// TwinCAT 3 PLC project RoboTelRuntime
// Company: Leibniz-Institut fuer Astrophysik Potsdam
// Author: Joerg Weingrill
// ProgramVersion: 3.1.4023.0
// libraries:
//   Tc2_Math, * (Beckhoff Automation GmbH)
//   Tc2_MC2, * (Beckhoff Automation GmbH)
//   Tc2_MC2_Drive, * (Beckhoff Automation GmbH)
//   Tc2_ModbusRTU, * (Beckhoff Automation GmbH)
//   Tc2_NC, * (Beckhoff Automation GmbH)
//   Tc2_Standard, * (Beckhoff Automation GmbH)
//   Tc2_System, * (Beckhoff Automation GmbH)
//   Tc2_Utilities, * (Beckhoff Automation GmbH)
//   Tc3_IotBase, * (Beckhoff Automation GmbH)
//   Tc3_Module, * (Beckhoff Automation GmbH)
//   PS_DcUpsEC,2.0,Phoenix Contact GmbH & Co.KG
// project tree:
//   DUTs/ E_TCSCommand.TcDUT, E_TCSErrors.TcDUT, E_TelescopeMode.TcDUT, ST_DomeStruct.TcDUT
//   / GlobalTextList.TcGTLO, PlcTask.TcTTO, Visualisierungsmanager.TcVMO (not stored)
//   GVLs/ GVL_Auxiliary.TcGVL, GVL_Dome.TcGVL, GVL_Environment.TcGVL, GVL_FilterWheel.TcGVL, GVL_pendant_control.TcGVL, GVL_Hydraulics.TcGVL, GVL_Safety.TcGVL, GVL_Telescope.TcGVL, GVL_Main.TcGVL
//   POUs/ AuxiliaryControl.TcPOU, CoverControl.TcPOU, DerotatorControl.TcPOU, DomeControl.TcPOU, DomeLowLevelControl.TcPOU, ElevationControl.TcPOU, AzimuthElevationControl.TcPOU, Environment.TcPOU, FanControl.TcPOU, FilterWheelControl.TcPOU, FocusControl.TcPOU, HydraulicsControl.TcPOU, MAIN.TcPOU, NasmythControl.TcPOU, PendantControl.TcPOU, SafetyHandling.TcPOU, TelescopeAuxiliary.TcPOU, TelescopeControl.TcPOU, Transformer.TcPOU
//   POUs/FunctionBlocks/ CO_ABERRATION.TcPOU, CO_REFRACT.TcPOU, FB_ALTAZ2HADEC.TcPOU, FB_AstroClock.TcPOU, FB_Axis2.TcPOU, FB_BLINK.TcPOU, FB_ButtonEnable.TcPOU, FB_CO_NUTATE.TcPOU, FB_EQ2HOR2.TcPOU, FB_EventLog.TcPOU, FB_HOR2EQ.TcPOU, FB_LightTimer.TcPOU, FB_MOONPOS.TcPOU, FB_MQTTCommunication.TcPOU, FB_NUTATE.TcPOU, FB_PRECESS.TcPOU, FB_SUNPOS.TcPOU, FB_TimeAverage.TcPOU, FB_Timer.TcPOU, FB_TONTP.TcPOU, FB_InfluxMessage.TcPOU, TIMER.TcPOU
//   POUs/Functions/ ATAN2.TcPOU, CO_REFRACT_FORWARD.TcPOU, CT2LST.TcPOU, DateTime2JD.TcPOU, F_Derotatorvelocity.TcPOU, F_Dewpoint.TcPOU, F_YREAL.TcPOU, F_DerotatorPosition2.TcPOU, LREAL_TO_FMTESTR.TcPOU, POLY.TcPOU, NCError_TO_STRING.TcPOU, TEN.TcPOU, Trigger.TcPOU
//   VISUs/ Visualization.TcVIS
// real-time tasks:
//   TASK PlcTask: cycle T#10ms, priority 14, ADS port 350
// motion (NC):
//   TASK NC-Task 1 SAF: cycle T#2ms, priority 4, ADS port 501
//   TASK NC-Task 1 SVB: cycle T#10ms, priority 8, ADS port 511
//   AXIS Focus (id 1)
//     Dynamic: AccelerationMaximum=100, DecelerationMaximum=100, Acceleration=2.47294, Deceleration=2.47294, Jerk=2.3521
//     Velo: RefSearch=0.2, RefSync=0.2, SlowManual=0.1, FastManual=0.5, Maximum=5
//     PositionAreaControl: Enable=false
//     TargetPosControl: Enable=false
//     OtherSettings: AllowMotionCmdToSlave=true, PulseDistancePos=1, PulseDistanceNeg=1
//     encoder EncType=4
//       EncPara: ScaleFactorNumerator=0.001, ScaleFactorDenominator=5, MaxCount=#x0000ffff
//         SoftEndMinControl: Enable=true
//         SoftEndMaxControl: Range=100
//         Inc: RefSoftSyncMask=#x0000ffff
//     drive DrvType=23
//       Analog: VeloReferenz=10.2713178, VeloScale=10, TorqueScale=10, ScaleFactorActTorque=10
//       TimeComp: TaskDelayCycles=1
//     controller CtrType=1
//       CtrPara: PriorControlFactor=0.1
//         PosDiffControl: Range=1
//         PID: PosKp=5
//         Observer: BandWidth=20
//   AXIS Derotator (id 7)
//     General: UnitName=°
//     Dynamic: AccelerationMaximum=10, DecelerationMaximum=10, Acceleration=5, Deceleration=5, Jerk=10
//     Velo: RefSearch=2, RefSync=2, SlowManual=1, FastManual=3, Fast=3.08588033040365, Maximum=3
//     PositionAreaControl: Enable=false
//     OtherSettings: AllowMotionCmdToSlave=true
//     encoder EncType=8
//       EncPara: ScaleFactorNumerator=0.1, ScaleFactorDenominator=1048576, MaxCount=#xffffffff
//         SoftEndMaxControl: Range=465
//         Inc: RefPosition=460
//     drive DrvType=9
//       DrvPara: MaxCount=#xffffffff, DriveControlDWord=#x00030100
//         Analog: VeloReferenz=3.39446836344401, VeloScale=1.02400649589962, ScaleFactorActTorque=0.1
//         TimeComp: TaskDelayCycles=1
//     controller CtrType=1
//       CtrPara: PriorControlFactor=1
//         PosDiffControl: Range=1
//         Observer: BandWidth=20
//   AXIS Azimuth (id 9)
//     General: UnitName=°
//     Dynamic: AccelerationMaximum=10, DecelerationMaximum=10, Acceleration=3.08, Deceleration=3.08, Jerk=1.75674
//     Velo: RefSearch=2, RefSync=2, SlowManual=1, FastManual=5, Fast=1663.37310791016, Maximum=10
//     OtherSettings: AllowMotionCmdToSlave=true
//     encoder EncType=8
//       EncPara: ScaleFactorNumerator=360, ScaleFactorDenominator=1048576, MaxCount=#xffffffff
//         SoftEndMinControl: Enable=true
//         SoftEndMaxControl: Enable=true, Range=450
//         Inc: RefPosition=156.1195, RefMode=2
//     drive DrvType=9
//       DrvPara: MaxCount=#xffffffff, DriveControlDWord=#x00030100
//         Analog: VeloReferenz=1188, VeloScale=1.02400649589962, ScaleFactorActTorque=0.1
//         TimeComp: TaskDelayCycles=1
//     controller CtrType=1
//       CtrPara: PriorControlFactor=1
//         PosDiffControl: Range=10
//         Observer: BandWidth=20
//   AXIS Elevation (id 10)
//     General: UnitName=°
//     Dynamic: AccelerationMaximum=2443.086, DecelerationMaximum=2443.086, Acceleration=3.24, Deceleration=3.24, Jerk=1.69316
//     Velo: RefSearch=0.5, RefSync=0.5, SlowManual=1, FastManual=3, Fast=1628.724, Maximum=10
//     OtherSettings: AllowMotionCmdToSlave=true
//     encoder EncType=8
//       EncPara: ScaleFactorNumerator=360, ScaleFactorDenominator=1048576, MaxCount=#xffffffff
//         SoftEndMinControl: Enable=true
//         SoftEndMaxControl: Enable=true, Range=91
//         Inc: RefPosition=45, RefMode=2
//     drive DrvType=9
//       DrvPara: MaxCount=#xffffffff, DriveControlDWord=#x00030100
//         Analog: VeloReferenz=1188, VeloScale=1.02400649589962, ScaleFactorActTorque=0.1
//         TimeComp: TaskDelayCycles=1
//     controller CtrType=1
//       CtrPara: PriorControlFactor=1
//         PosDiffControl: Range=10
//         Observer: BandWidth=20
//   AXIS DomeAzimuth (id 2)
//     General: UnitName=°, UnitFlags=#x00000004
//     Dynamic: AccelerationMaximum=1, DecelerationMaximum=1
//     Velo: RefSearch=15, RefSync=15, SlowManual=25, FastManual=75, Fast=100, Maximum=100
//     PositionAreaControl: Enable=false
//     TargetPosControl: Range=10
//     OtherSettings: AllowMotionCmdToSlave=true
//     Discrete: CreepDistancePos=10, CreepDistanceNeg=10, BreakDistancePos=2.5, BreakDistanceNeg=2.5, BreakDelayPos=0.1, BreakDelayNeg=0.1, CreepDistanceStop=5
//     encoder EncType=4
//       EncPara: ScaleFactorNumerator=0.0003641, Inverse=true, MaxCount=#x0000ffff
//         Inc: RefSearchInverse=true, RefPosition=172.5, RefMode=2, RefSoftSyncMask=#x0000ffff
//     drive DrvType=7
//       Analog: TorqueScale=10, ScaleFactorActTorque=0.1
//       TimeComp: TaskDelayCycles=1
//     controller CtrType=7
//       CtrPara: PriorControlFactor=1
//         PosDiffControl: Range=10
//         Observer: BandWidth=20
//   AXIS Filterrad (id 3)
//     General: UnitName=°, UnitFlags=#x00000004
//     Dynamic: Acceleration=155.749978166623, Deceleration=155.749978166623, Jerk=467.249868999747
//     Velo: RefSearch=1.03833333333333, RefSync=1.03833333333333, SlowManual=5.19166666666667, FastManual=31.15, Fast=103.833333333333, Maximum=103.833
//     OtherSettings: AllowMotionCmdToSlave=true
//     encoder EncType=19
//       EncPara: ScaleFactorNumerator=5, ScaleFactorDenominator=1048576, MaxCount=#xffffffff
//     drive DrvType=16
//       DrvPara: MaxCount=#xffffffff, DriveControlDWord=#x00020000
//         Analog: VeloReferenz=114.216666666667, VeloScale=32, TorqueScale=10, ScaleFactorActTorque=0.1
//         TimeComp: TaskDelayCycles=1
//     controller CtrType=1
//       CtrPara: PriorControlFactor=1
//         PosDiffControl: Enable=false
//         Observer: BandWidth=20
// I/O:
//   DEVICE Gerät 1 (EtherCAT), AmsNetId 5.78.96.50.2.1
//     Klemme 1 (EK1200) [EK1200-5000 EtherCAT Netzteil (2A E-Bus)] // Hauptschrank
//       TwinSAFE Logic (EL6910) [EL6910, TwinSAFE PLC]
//       TwinSAFE IN (EL1904) [EL1904, 4 K. Safety Eingang 24V, TwinSAFE]
//         modules: Module 1 (FSOES)
//       TwinSAFE OUT (EL2904) [EL2904, 4 K. Safety Ausgang 24V, 0.5A, TwinSAFE]
//         modules: Module 1 (FSOES), Module 2 (DO)
//       Power Diag (EL3443) [EL3443 3K. Leistungsmessung]
//       Klemme 29 (EL9410) [EL9410 E-Bus Netzteilklemme (Diagnose)]
//       Panel IN (EL1008) [EL1008 8K. Dig. Eingang 24V, 3ms] // Main panel
//       Hydraulik IN (EL1008) [EL1008 8K. Dig. Eingang 24V, 3ms] // Ölstatus
//       Aux IN (EL1008) [EL1008 8K. Dig. Eingang 24V, 3ms]
//       Panel OUT (EL2008) [EL2008 8K. Dig. Ausgang 24V, 0.5A]
//       Hydraulics OUT (EL2008) [EL2008 8K. Dig. Ausgang 24V, 0.5A]
//       Cabinet TEMP (EL3202-0010) [EL3202-0010 2K. Ana. Eingang PT100 (RTD), hochgenau]
//       Klemme 7 (EK1521) [EK1521 1-Port EtherCAT-Abzweig (FX-MultiMode)]
//         Telescope Cabinet (EK1501) [EK1501 EtherCAT-Koppler (2A E-Bus, FX-MultiMode, ID-Switch)] // Unterverteiler Teleskop
//           Handcontrol IN1 (EL1008) [EL1008 8K. Dig. Eingang 24V, 3ms]
//           Handcontrol IN2 (EL1008) [EL1008 8K. Dig. Eingang 24V, 3ms]
//           Limits IN1 (EL1008) [EL1008 8K. Dig. Eingang 24V, 3ms]
//           Cover IN (EL1008) [EL1008 8K. Dig. Eingang 24V, 3ms]
//           Hydraulics IN (EL1008) [EL1008 8K. Dig. Eingang 24V, 3ms]
//           Handcontrol OUT (EL2008) [EL2008 8K. Dig. Ausgang 24V, 0.5A]
//           Aux OUT (EL2008) [EL2008 8K. Dig. Ausgang 24V, 0.5A] // brakes and horn
//           Temp2 (EL3202-0010) [EL3202-0010 2K. Ana. Eingang PT100 (RTD), hochgenau]
//           Temp4 (EL3202-0010) [EL3202-0010 2K. Ana. Eingang PT100 (RTD), hochgenau]
//           Power (EL9410) [EL9410 E-Bus Netzteilklemme (Diagnose)]
//           Motor1 (EL7342) [EL7342 2K. DC-Motor-Endstufe (50V, 3.5A)] // Focus
//           Encoder (EL5101) [EL5101 1K. Inc. Encoder 5V] // Fokus Encoder
//           M3 (EL2042) [EL2042 2K. Dig. Ausgang 24V, 4A]
//           Cover2 (EL2042) [EL2042 2K. Dig. Ausgang 24V, 4A]
//           Cover3 (EL2042) [EL2042 2K. Dig. Ausgang 24V, 4A]
//           Klemme 27 (EL9011) [EL9011 Endklemme]
//         Dome Azimuth (EK1501) [EK1501 EtherCAT-Koppler (2A E-Bus, FX-MultiMode, ID-Switch)]
//           Dome IN (EL1008) [EL1008 8K. Dig. Eingang 24V, 3ms]
//           Dome OUT (EL2008) [EL2008 8K. Dig. Ausgang 24V, 0.5A]
//           Velo IN (EL3064) [EL3064 4K.Ana. Eingang 0-10V]
//           Velo OUT (EL4002) [EL4002 2K. Ana. Ausgang 0-10V, 12bit]
//           Encoder (EL5151) [EL5151 1K. Inc. Encoder]
//           Analog IN (EL3024) [EL3024 4K. Ana. Eingang 4-20mA DIFF]
//           Klemme 70 (EL9011) [EL9011 Endklemme]
//         Weather (EK1501) [EK1501 EtherCAT-Koppler (2A E-Bus, FX-MultiMode, ID-Switch)]
//           Analog IN (EL3068) [EL3068 8K. Ana. Eingang 0-10V]
//           Rain IN (EL1008) [EL1008 8K. Dig. Eingang 24V, 3ms]
//           Klemme 93 (EL6021) [EL6021 Schnittstelle (RS422/485)]
//           Klemme 80 (EL9011) [EL9011 Endklemme]
//       Klemme 84 (EK1521) [EK1521 1-Port EtherCAT-Abzweig (FX-MultiMode)]
//         Filterwheel Cabinet (EK1501) [EK1501 EtherCAT-Koppler (2A E-Bus, FX-MultiMode, ID-Switch)]
//           Filterrad (EL7211-0010) [EL7211-0010 1K. MDP742 Servo-Motor-Endstufe mit OCT (50V, 4,5A RMS)]
//             startup 32784:18 := 0500
//             startup 32784:19 := 4C01
//             startup 32784:20 := 96000000
//             startup 32784:21 := 62000000
//             startup 32785:17 := 68420000
//             startup 32785:18 := A00F0000
//             startup 32785:19 := 03
//             startup 32785:21 := 0E01
//             startup 32785:22 := 7D000000
//             startup 32785:24 := 8B000000
//             startup 32785:25 := 1C00
//             startup 32785:27 := DE040000
//             startup 32785:45 := 3402
//           Klemme 89 (EL1008) [EL1008 8K. Dig. Eingang 24V, 3ms]
//           Klemme 90 (EL2008) [EL2008 8K. Dig. Ausgang 24V, 0.5A]
//           Serial IO (EL6001) [EL6001 Schnittstelle (RS232)]
//           Klemme 24 (EL3064) [EL3064 4K.Ana. Eingang 0-10V]
//           Klemme 101 (EL9011) [EL9011 Endklemme]
//       Klemme 22 (EK1110) [EK1110 EtherCAT-Verlängerung]
//     Box 107 (Uninterruptible Power Supply) [QUINT4-UPS/24DC/24DC/40/EC]
//     Derotator (AX5206-0000-0213) [AX5206-0000-0213 EtherCAT Drive (SoE, 2 Ch.)]
//     Azimuth (AX5125-0000-0213) [AX5125-0000-0213 EtherCAT Drive (SoE, 1 Ch.)] // Azimut
//     Elevation (AX5125-0000-0213) [AX5125-0000-0213 EtherCAT Drive (SoE, 1 Ch.)] // Elevation
// variable links:
//   Device 1 (EtherCAT) <-> Device 1 (EtherCAT)/Term 1 (EK1200)/TwinSAFE IN (EL1904)
//     Term 1 (EK1200)/TwinSAFE Logic (EL6910)/ConnectionOutputs/TwinSafeGroup1.Klemme 30 (EL1904) - Module 1 (FSOES)_2 RxPDO <-> Module 1 (FSOES)/TxPDO/FSOE
//   Device 1 (EtherCAT) <-> Device 1 (EtherCAT)/Term 1 (EK1200)/TwinSAFE Logic (EL6910)
//     Term 1 (EK1200)/TwinSAFE IN (EL1904)/Module 1 (FSOES)/RxPDO/FSOE <-> ConnectionInputs/TwinSafeGroup1.Klemme 30 (EL1904) - Module 1 (FSOES)_2 TxPDO
//     Term 1 (EK1200)/TwinSAFE OUT (EL2904)/Module 1 (FSOES)/TxPDO/FSOE <-> ConnectionOutputs/TwinSafeGroup1.Klemme 31 (EL2904) - Module 1 (FSOES)_3 RxPDO
//   Device 1 (EtherCAT) <-> Device 1 (EtherCAT)/Term 1 (EK1200)/TwinSAFE OUT (EL2904)
//     Term 1 (EK1200)/TwinSAFE Logic (EL6910)/ConnectionInputs/TwinSafeGroup1.Klemme 31 (EL2904) - Module 1 (FSOES)_3 TxPDO <-> Module 1 (FSOES)/RxPDO/FSOE
//   NC-Task 1 SAF/Axes/Azimuth <-> Device 1 (EtherCAT)/Azimuth (AX5125-0000-0213)
//     Drive/Inputs/In/nDataIn1 <-> AT/Following distance
//     Drive/Inputs/In/nDcOutputTime <-> InfoData/DcOutputShift
//     Drive/Inputs/In/nState1 <-> AT/Drive status word @bit 8
//     Drive/Inputs/In/nState2 <-> AT/Drive status word
//     Drive/Inputs/In/nState4 @bit 1 <-> WcState/InputToggle
//     Drive/Inputs/In/nState4 <-> WcState/WcState
//     Drive/Outputs/Out/nCtrl1 <-> MDT/Master control word @bit 8
//     Drive/Outputs/Out/nDataOut1 <-> MDT/Position command value
//     Enc/Inputs/In/nDataIn1 <-> AT/Position feedback 1 value
//     Enc/Inputs/In/nDataIn3 <-> AT/Probe value 1 positive edge
//     Enc/Inputs/In/nDcInputTime <-> InfoData/DcInputShift
//     Enc/Inputs/In/nState4 @bit 1 <-> WcState/InputToggle
//     Enc/Inputs/In/nState4 <-> WcState/WcState
//     Enc/Inputs/In/nState5 <-> AT/Probe 1 positive latched
//     Enc/Outputs/Out/nCtrl5 <-> MDT/Probe 1 enable
//   NC-Task 1 SAF/Axes/Derotator <-> Device 1 (EtherCAT)/Derotator (AX5206-0000-0213)
//     Drive/Inputs/In/nDataIn1 <-> AT 1/Following distance
//     Drive/Inputs/In/nDcOutputTime <-> InfoData/DcOutputShift
//     Drive/Inputs/In/nState1 <-> AT 1/Drive status word @bit 8
//     Drive/Inputs/In/nState2 <-> AT 1/Drive status word
//     Drive/Inputs/In/nState4 @bit 1 <-> WcState/InputToggle
//     Drive/Inputs/In/nState4 <-> WcState/WcState
//     Drive/Outputs/Out/nCtrl1 <-> MDT 1/Master control word @bit 8
//     Drive/Outputs/Out/nDataOut1 <-> MDT 1/Position command value
//     Enc/Inputs/In/nDataIn1 <-> AT 1/Position feedback 1 value
//     Enc/Inputs/In/nDcInputTime <-> InfoData/DcInputShift
//     Enc/Inputs/In/nState4 @bit 1 <-> WcState/InputToggle
//     Enc/Inputs/In/nState4 <-> WcState/WcState
//   NC-Task 1 SAF/Axes/DomeAzimuth <-> Device 1 (EtherCAT)/Term 1 (EK1200)/Term 7 (EK1521)/Dome Azimuth (EK1501)/Encoder (EL5151)
//     Enc/Inputs/In/nDataIn1[0] <-> ENC Inputs/Counter value
//     Enc/Inputs/In/nDataIn2[0] <-> ENC Inputs/Latch value
//     Enc/Inputs/In/nState1 @bit 7 <-> ENC Inputs/Status/Extrapolation stall
//     Enc/Inputs/In/nState1 <-> ENC Inputs/Status/Latch C valid
//     Enc/Inputs/In/nState1 @bit 1 <-> ENC Inputs/Status/Latch extern valid
//     Enc/Inputs/In/nState1 @bit 2 <-> ENC Inputs/Status/Set counter done
//     Enc/Inputs/In/nState2 @bit 4 <-> ENC Inputs/Status/Status of extern latch
//     Enc/Inputs/In/nState2 <-> ENC Inputs/Status/Status of input A
//     Enc/Inputs/In/nState2 @bit 1 <-> ENC Inputs/Status/Status of input B
//     Enc/Inputs/In/nState2 @bit 2 <-> ENC Inputs/Status/Status of input C
//     Enc/Inputs/In/nState2 @bit 5 <-> ENC Inputs/Status/Sync error
//     Enc/Inputs/In/nState2 @bit 7 <-> ENC Inputs/Status/TxPDO Toggle
//     Enc/Inputs/In/nState4 @bit 1 <-> WcState/InputToggle
//     Enc/Inputs/In/nState4 <-> WcState/WcState
//     Enc/Outputs/Out/nCtrl1 <-> ENC Outputs/Control/Enable latch C
//     Enc/Outputs/Out/nCtrl1 @bit 3 <-> ENC Outputs/Control/Enable latch extern on negative edge
//     Enc/Outputs/Out/nCtrl1 @bit 1 <-> ENC Outputs/Control/Enable latch extern on positive edge
//     Enc/Outputs/Out/nCtrl1 @bit 2 <-> ENC Outputs/Control/Set counter
//     Enc/Outputs/Out/nDataOut1[0] <-> ENC Outputs/Set counter value
//   NC-Task 1 SAF/Axes/Elevation <-> Device 1 (EtherCAT)/Elevation (AX5125-0000-0213)
//     Drive/Inputs/In/nDataIn1 <-> AT/Following distance
//     Drive/Inputs/In/nDcOutputTime <-> InfoData/DcOutputShift
//     Drive/Inputs/In/nState1 <-> AT/Drive status word @bit 8
//     Drive/Inputs/In/nState2 <-> AT/Drive status word
//     Drive/Inputs/In/nState4 @bit 1 <-> WcState/InputToggle
//     Drive/Inputs/In/nState4 <-> WcState/WcState
//     Drive/Outputs/Out/nCtrl1 <-> MDT/Master control word @bit 8
//     Drive/Outputs/Out/nDataOut1 <-> MDT/Position command value
//     Enc/Inputs/In/nDataIn1 <-> AT/Position feedback 1 value
//     Enc/Inputs/In/nDataIn3 <-> AT/Probe value 1 positive edge
//     Enc/Inputs/In/nDcInputTime <-> InfoData/DcInputShift
//     Enc/Inputs/In/nState4 @bit 1 <-> WcState/InputToggle
//     Enc/Inputs/In/nState4 <-> WcState/WcState
//     Enc/Inputs/In/nState5 <-> AT/Probe 1 positive latched
//     Enc/Outputs/Out/nCtrl5 <-> MDT/Probe 1 enable
//   NC-Task 1 SAF/Axes/Filterrad <-> Device 1 (EtherCAT)/Term 1 (EK1200)/Term 84 (EK1521)/Filterwheel Cabinet (EK1501)/Filterrad (EL7211-0010)
//     Drive/Inputs/In/nDcOutputTime <-> InfoData/DcOutputShift
//     Drive/Inputs/In/nState1 <-> DRV Statusword/Statusword
//     Drive/Inputs/In/nState2 <-> DRV Statusword/Statusword @bit 8
//     Drive/Inputs/In/nState4 @bit 1 <-> WcState/InputToggle
//     Drive/Inputs/In/nState4 <-> WcState/WcState
//     Drive/Outputs/Out/nCtrl1 <-> DRV Controlword/Controlword
//     Drive/Outputs/Out/nCtrl2 <-> DRV Controlword/Controlword @bit 8
//     Drive/Outputs/Out/nDataOut2 <-> DRV Target velocity/Target velocity
//     Enc/Inputs/In/nDataIn1 <-> FB Position/Position
//     Enc/Inputs/In/nDataIn3 <-> FB Touch probe 1 pos position/TP1 Pos position
//     Enc/Inputs/In/nDataIn5 <-> FB Touch probe 2 pos position/TP2 Pos position
//     Enc/Inputs/In/nDataIn4 <-> FB Touch probe 1 neg position/TP1 Neg position
//     Enc/Inputs/In/nDataIn6 <-> FB Touch probe 2 neg position/TP2 Neg position
//     Enc/Inputs/In/nDcInputTime <-> InfoData/DcInputShift
//     Enc/Inputs/In/nState4 @bit 1 <-> WcState/InputToggle
//     Enc/Inputs/In/nState4 <-> WcState/WcState
//     Enc/Inputs/In/nState5 <-> FB Touch probe status/Touch probe status/TP1 Enable
//     Enc/Inputs/In/nState6 <-> FB Touch probe status/Touch probe status/TP2 Enable
//     Enc/Inputs/In/nState5 @bit 7 <-> FB Touch probe status/Touch probe status/TP1 Input
//     Enc/Inputs/In/nState6 @bit 7 <-> FB Touch probe status/Touch probe status/TP2 Input
//     Enc/Inputs/In/nState5 @bit 2 <-> FB Touch probe status/Touch probe status/TP1 Neg value stored
//     Enc/Inputs/In/nState6 @bit 2 <-> FB Touch probe status/Touch probe status/TP2 Neg value stored
//     Enc/Inputs/In/nState5 @bit 1 <-> FB Touch probe status/Touch probe status/TP1 Pos value stored
//     Enc/Inputs/In/nState6 @bit 1 <-> FB Touch probe status/Touch probe status/TP2 Pos value stored
//     Enc/Outputs/Out/nCtrl5 @bit 1 <-> FB Touch probe control/Touch probe function/TP1 Continous
//     Enc/Outputs/Out/nCtrl6 @bit 1 <-> FB Touch probe control/Touch probe function/TP2 Continous
//     Enc/Outputs/Out/nCtrl5 <-> FB Touch probe control/Touch probe function/TP1 Enable
//     Enc/Outputs/Out/nCtrl6 <-> FB Touch probe control/Touch probe function/TP2 Enable
//     Enc/Outputs/Out/nCtrl5 @bit 5 <-> FB Touch probe control/Touch probe function/TP1 Enable neg edge
//     Enc/Outputs/Out/nCtrl6 @bit 5 <-> FB Touch probe control/Touch probe function/TP2 Enable neg edge
//     Enc/Outputs/Out/nCtrl5 @bit 4 <-> FB Touch probe control/Touch probe function/TP1 Enable pos edge
//     Enc/Outputs/Out/nCtrl6 @bit 4 <-> FB Touch probe control/Touch probe function/TP2 Enable pos edge
//     Enc/Outputs/Out/nCtrl5 @bit 2 <-> FB Touch probe control/Touch probe function/TP1 Trigger mode
//     Enc/Outputs/Out/nCtrl6 @bit 2 <-> FB Touch probe control/Touch probe function/TP2 Trigger mode
//   NC-Task 1 SAF/Axes/Focus <-> Device 1 (EtherCAT)/Term 1 (EK1200)/Term 7 (EK1521)/Telescope Cabinet (EK1501)/Encoder (EL5101)
//     Enc/Inputs/In/nDataIn1[0] <-> ENC Status compact/Counter value
//     Enc/Inputs/In/nDataIn2[0] <-> ENC Status compact/Latch value
//     Enc/Inputs/In/nState1 @bit 4 <-> ENC Status compact/Status/Counter overflow
//     Enc/Inputs/In/nState1 @bit 3 <-> ENC Status compact/Status/Counter underflow
//     Enc/Inputs/In/nState1 @bit 7 <-> ENC Status compact/Status/Extrapolation stall
//     Enc/Inputs/In/nState1 <-> ENC Status compact/Status/Latch C valid
//     Enc/Inputs/In/nState1 @bit 1 <-> ENC Status compact/Status/Latch extern valid
//     Enc/Inputs/In/nState1 @bit 6 <-> ENC Status compact/Status/Open circuit
//     Enc/Inputs/In/nState1 @bit 2 <-> ENC Status compact/Status/Set counter done
//     Enc/Inputs/In/nState1 @bit 5 <-> ENC Status compact/Status/Status of input status
//     Enc/Inputs/In/nState2 @bit 4 <-> ENC Status compact/Status/Status of extern latch
//     Enc/Inputs/In/nState2 <-> ENC Status compact/Status/Status of input A
//     Enc/Inputs/In/nState2 @bit 1 <-> ENC Status compact/Status/Status of input B
//     Enc/Inputs/In/nState2 @bit 2 <-> ENC Status compact/Status/Status of input C
//     Enc/Inputs/In/nState2 @bit 3 <-> ENC Status compact/Status/Status of input gate
//     Enc/Inputs/In/nState2 @bit 5 <-> ENC Status compact/Status/Sync error
//     Enc/Inputs/In/nState2 @bit 6 <-> ENC Status compact/Status/TxPDO State
//     Enc/Inputs/In/nState2 @bit 7 <-> ENC Status compact/Status/TxPDO Toggle
//     Enc/Inputs/In/nState4 @bit 1 <-> WcState/InputToggle
//     Enc/Inputs/In/nState4 <-> WcState/WcState
//     Enc/Outputs/Out/nCtrl1 <-> ENC Control compact/Control/Enable latch C
//     Enc/Outputs/Out/nCtrl1 @bit 3 <-> ENC Control compact/Control/Enable latch extern on negative edge
//     Enc/Outputs/Out/nCtrl1 @bit 1 <-> ENC Control compact/Control/Enable latch extern on positive edge
//     Enc/Outputs/Out/nCtrl1 @bit 2 <-> ENC Control compact/Control/Set counter
//     Enc/Outputs/Out/nDataOut1[0] <-> ENC Control compact/Set counter value
//   NC-Task 1 SAF/Axes/Focus <-> Device 1 (EtherCAT)/Term 1 (EK1200)/Term 7 (EK1521)/Telescope Cabinet (EK1501)/Motor1 (EL7342)
//     Drive/Inputs/In/nState1 @bit 3 <-> DCM Status Channel 1/Status/Error
//     Drive/Inputs/In/nState1 @bit 5 <-> DCM Status Channel 1/Status/Moving negative
//     Drive/Inputs/In/nState1 @bit 4 <-> DCM Status Channel 1/Status/Moving positive
//     Drive/Inputs/In/nState1 @bit 1 <-> DCM Status Channel 1/Status/Ready
//     Drive/Inputs/In/nState1 <-> DCM Status Channel 1/Status/Ready to enable
//     Drive/Inputs/In/nState1 @bit 6 <-> DCM Status Channel 1/Status/Torque reduced
//     Drive/Inputs/In/nState1 @bit 2 <-> DCM Status Channel 1/Status/Warning
//     Drive/Inputs/In/nState2 @bit 3 <-> DCM Status Channel 1/Status/Digital input 1
//     Drive/Inputs/In/nState2 @bit 4 <-> DCM Status Channel 1/Status/Digital input 2
//     Drive/Inputs/In/nState2 @bit 5 <-> DCM Status Channel 1/Status/Sync error
//     Drive/Inputs/In/nState2 @bit 7 <-> DCM Status Channel 1/Status/TxPDO Toggle
//     Drive/Inputs/In/nState4 @bit 1 <-> WcState/InputToggle
//     Drive/Inputs/In/nState4 <-> WcState/WcState
//     Drive/Outputs/Out/nCtrl1 <-> DCM Control Channel 1/Control/Enable
//     Drive/Outputs/Out/nCtrl1 @bit 2 <-> DCM Control Channel 1/Control/Reduce torque
//     Drive/Outputs/Out/nCtrl1 @bit 1 <-> DCM Control Channel 1/Control/Reset
//     Drive/Outputs/Out/nDataOut2[0] <-> DCM Velocity Channel 1/Velocity
//   RoboTelRuntime/RoboTelRuntime Instance <-> Device 1 (EtherCAT)/Azimuth (AX5125-0000-0213)
//     PlcTask Inputs/GVL_Telescope.Azimuth_diagnostic <-> AT/Diagnostic number
//     PlcTask Inputs/GVL_Telescope.Azimuth_inputs <-> AT/Digital inputs, state
//     PlcTask Inputs/GVL_Telescope.Azimuth_torque <-> AT/Torque/force feedback value
//   RoboTelRuntime/RoboTelRuntime Instance <-> Device 1 (EtherCAT)/Box 107 (Uninterruptible Power Supply)
//     PlcTask Inputs/MAIN.arrInputPD @bit {304..432 step 32} <-> TxPDO 1/BATTERY {1..5} ALARMS  (5 links)
//     PlcTask Inputs/MAIN.arrInputPD @bit 464 <-> TxPDO 1/QUINT CHARGER ALARMS
//     PlcTask Inputs/MAIN.arrInputPD @bit 80 <-> TxPDO 1/STATUS ACTUAL INPUT CURRENT
//     PlcTask Inputs/MAIN.arrInputPD @bit 64 <-> TxPDO 1/STATUS ACTUAL INPUT VOLTAGE
//     PlcTask Inputs/MAIN.arrInputPD @bit 112 <-> TxPDO 1/STATUS ACTUAL OUTPUT CURRENT 1
//     PlcTask Inputs/MAIN.arrInputPD @bit 96 <-> TxPDO 1/STATUS ACTUAL OUTPUT VOLTAGE 1
//     PlcTask Inputs/MAIN.arrInputPD @bit 128 <-> TxPDO 1/STATUS BATTERY ACTUAL VOLTAGE
//     PlcTask Inputs/MAIN.arrInputPD @bit 144 <-> TxPDO 1/STATUS BATTERY CHARGE CURRENT
//     PlcTask Inputs/MAIN.arrInputPD @bit 160 <-> TxPDO 1/STATUS BATTERY TEMPERATURE
//     PlcTask Inputs/MAIN.arrInputPD @bit 176 <-> TxPDO 1/STATUS DEVICE TEMPERATURE
//     PlcTask Inputs/MAIN.arrInputPD <-> TxPDO 1/STATUS FUNCTIONS
//     PlcTask Inputs/MAIN.arrInputPD @bit 32 <-> TxPDO 1/STATUS INTERFACE
//     PlcTask Inputs/MAIN.arrInputPD @bit 192 <-> TxPDO 1/STATUS SOC REMAINING TIME
//     PlcTask Inputs/MAIN.arrInputPD @bit 224 <-> TxPDO 1/STATUS SOC REMAINING TIME PC SHUTDOWN
//     PlcTask Inputs/MAIN.arrInputPD @bit 240 <-> TxPDO 1/STATUS SOH REMAINING LIFETIME
//     PlcTask Inputs/MAIN.arrInputPD @bit 272 <-> TxPDO 1/UPS DIAGNOSIS ALARMS
//     PlcTask Inputs/MAIN.arrInputPD @bit 256 <-> TxPDO 1/UPS PROCESS ALARMS
//   RoboTelRuntime/RoboTelRuntime Instance <-> Device 1 (EtherCAT)/Derotator (AX5206-0000-0213)
//     PlcTask Inputs/GVL_Telescope.Derotator_inputs <-> AT 1/Digital inputs, state
//     PlcTask Inputs/GVL_Telescope.Derotator_torque <-> AT 1/Torque/force feedback value
//   RoboTelRuntime/RoboTelRuntime Instance <-> Device 1 (EtherCAT)/Elevation (AX5125-0000-0213)
//     PlcTask Inputs/GVL_Telescope.Elevation_diagnostic <-> AT/Diagnostic number
//     PlcTask Inputs/GVL_Telescope.Elevation_inputs <-> AT/Digital inputs, state
//     PlcTask Inputs/GVL_Telescope.Elevation_torque <-> AT/Torque/force feedback value
//   RoboTelRuntime/RoboTelRuntime Instance <-> Device 1 (EtherCAT)/Term 1 (EK1200)/Aux IN (EL1008)
//     PlcTask Inputs/GVL_Main.brake_clearing <-> Channel 3/GVL_Main.brake_clearing
//     PlcTask Inputs/GVL_Main.phase_available <-> Channel 1/GVL_Main.phase_available
//     PlcTask Inputs/GVL_Main.power_available <-> Channel 2/GVL_Main.power_available
//   RoboTelRuntime/RoboTelRuntime Instance <-> Device 1 (EtherCAT)/Term 1 (EK1200)/Cabinet TEMP (EL3202-0010)
//     PlcTask Inputs/GVL_Main.main_cabinet_temperature <-> RTD Inputs Channel 1/GVL_Main.main_cabinet_temperature
//   RoboTelRuntime/RoboTelRuntime Instance <-> Device 1 (EtherCAT)/Term 1 (EK1200)/Hydraulics OUT (EL2008)
//     PlcTask Outputs/GVL_Hydraulics.oil_pump_enable <-> Channel 1/GVL_Hydraulics.oil_pump_enable
//     PlcTask Outputs/GVL_Hydraulics.oil_suction_enable <-> Channel 2/GVL_Hydraulics.oil_suction_enable
//     PlcTask Outputs/GVL_Main.softstart_trafo <-> Channel 7/GVL_Main.softstart_trafo
//     PlcTask Outputs/GVL_Telescope.brake_azimuth_eve <-> Channel 3/GVL_Telescope.brake_azimuth_eve
//   RoboTelRuntime/RoboTelRuntime Instance <-> Device 1 (EtherCAT)/Term 1 (EK1200)/Hydraulik IN (EL1008)
//     PlcTask Inputs/GVL_Hydraulics.oil_high <-> Channel 2/GVL_Hydraulics.oil_high
//     PlcTask Inputs/GVL_Hydraulics.oil_low <-> Channel 1/GVL_Hydraulics.oil_low
//     PlcTask Inputs/GVL_Hydraulics.oil_overtemperature <-> Channel 4/GVL_Hydraulics.oil_overtemperature
//     PlcTask Inputs/GVL_Hydraulics.oil_pressure_OK <-> Channel 3/GVL_Hydraulics.oil_pressure_OK
//     PlcTask Inputs/GVL_Hydraulics.oil_undertemperature <-> Channel 5/GVL_Hydraulics.oil_undertemperature
//     PlcTask Inputs/GVL_Hydraulics.oilfilter_dirty <-> Channel 6/GVL_Hydraulics.oilfilter_dirty
//     PlcTask Inputs/GVL_Hydraulics.pump_running <-> Channel 7/GVL_Hydraulics.pump_running
//     PlcTask Inputs/GVL_Hydraulics.suction_running <-> Channel 8/GVL_Hydraulics.suction_running
//   RoboTelRuntime/RoboTelRuntime Instance <-> Device 1 (EtherCAT)/Term 1 (EK1200)/Panel IN (EL1008)
//     PlcTask Inputs/GVL_Main.key_switch_remote <-> Channel 1/GVL_Main.key_switch_remote
//     PlcTask Inputs/GVL_Main.reset_switch <-> Channel 4/GVL_Main.reset_switch
//     PlcTask Inputs/GVL_Main.start_switch <-> Channel 2/GVL_Main.start_switch
//     PlcTask Inputs/GVL_Main.stop_switch <-> Channel 3/GVL_Main.stop_switch
//   RoboTelRuntime/RoboTelRuntime Instance <-> Device 1 (EtherCAT)/Term 1 (EK1200)/Panel OUT (EL2008)
//     PlcTask Outputs/GVL_Main.lamp_error <-> Channel 3/GVL_Main.lamp_error
//     PlcTask Outputs/GVL_Main.lamp_power <-> Channel 1/GVL_Main.lamp_power
//     PlcTask Outputs/GVL_Main.lamp_ready <-> Channel 2/GVL_Main.lamp_ready
//   RoboTelRuntime/RoboTelRuntime Instance <-> Device 1 (EtherCAT)/Term 1 (EK1200)/Power Diag (EL3443)
//     PlcTask Inputs/GVL_Main.L1_L2_Voltage <-> Total L-L Voltage/GVL_Main.L1_L2_Voltage
//     PlcTask Inputs/GVL_Main.L2_L3_Voltage <-> Total L-L Voltage/GVL_Main.L2_L3_Voltage
//     PlcTask Inputs/GVL_Main.L3_L1_Voltage <-> Total L-L Voltage/GVL_Main.L3_L1_Voltage
//   RoboTelRuntime/RoboTelRuntime Instance <-> Device 1 (EtherCAT)/Term 1 (EK1200)/Term 7 (EK1521)/Dome Azimuth (EK1501)/Analog IN (EL3024)
//     PlcTask Inputs/GVL_Environment.rawHumidityDome <-> AI Standard Channel 1/GVL_Environment.rawHumidityDome
//     PlcTask Inputs/GVL_Environment.rawTemperatureDome <-> AI Standard Channel 2/GVL_Environment.rawTemperatureDome
//   RoboTelRuntime/RoboTelRuntime Instance <-> Device 1 (EtherCAT)/Term 1 (EK1200)/Term 7 (EK1521)/Dome Azimuth (EK1501)/Dome IN (EL1008)
//     PlcTask Inputs/GVL_Dome.Azimuth_home <-> Channel 4/GVL_Dome.Azimuth_home
//     PlcTask Inputs/GVL_Dome.Clockwise <-> Channel 2/GVL_Dome.Clockwise
//     PlcTask Inputs/GVL_Dome.CounterClockwise <-> Channel 1/GVL_Dome.CounterClockwise
//   RoboTelRuntime/RoboTelRuntime Instance <-> Device 1 (EtherCAT)/Term 1 (EK1200)/Term 7 (EK1521)/Dome Azimuth (EK1501)/Dome OUT (EL2008)
//     PlcTask Outputs/GVL_Dome.DeHumidifier <-> Channel 5/GVL_Dome.DeHumidifier
//     PlcTask Outputs/GVL_Dome.Inverter_DirectionMinus <-> Channel 2/GVL_Dome.Inverter_DirectionMinus
//     PlcTask Outputs/GVL_Dome.Inverter_Enable <-> Channel 1/GVL_Dome.Inverter_Enable
//     PlcTask Outputs/GVL_Dome.Light <-> Channel 4/GVL_Dome.Light
//   RoboTelRuntime/RoboTelRuntime Instance <-> Device 1 (EtherCAT)/Term 1 (EK1200)/Term 7 (EK1521)/Dome Azimuth (EK1501)/Velo OUT (EL4002)
//     PlcTask Outputs/GVL_Dome.Inverter_Velocity <-> AO Outputs Channel 1/GVL_Dome.Inverter_Velocity
//   RoboTelRuntime/RoboTelRuntime Instance <-> Device 1 (EtherCAT)/Term 1 (EK1200)/Term 7 (EK1521)/Telescope Cabinet (EK1501)/Aux OUT (EL2008)
//     PlcTask Outputs/GVL_Telescope.focus_unlock <-> Channel 1/GVL_Telescope.focus_unlock
//     PlcTask Outputs/GVL_Telescope.horn <-> Channel 3/GVL_Telescope.horn
//     PlcTask Outputs/GVL_Telescope.nasmyth_lock <-> Channel 2/GVL_Telescope.nasmyth_lock
//   RoboTelRuntime/RoboTelRuntime Instance <-> Device 1 (EtherCAT)/Term 1 (EK1200)/Term 7 (EK1521)/Telescope Cabinet (EK1501)/Cover IN (EL1008)
//     PlcTask Inputs/GVL_Telescope.cover2_closed <-> Channel 4/GVL_Telescope.cover2_closed
//     PlcTask Inputs/GVL_Telescope.cover3_closed <-> Channel 6/GVL_Telescope.cover3_closed
//     PlcTask Inputs/GVL_Telescope.cover2_open <-> Channel 3/GVL_Telescope.cover2_open
//     PlcTask Inputs/GVL_Telescope.cover3_open <-> Channel 5/GVL_Telescope.cover3_open
//   RoboTelRuntime/RoboTelRuntime Instance <-> Device 1 (EtherCAT)/Term 1 (EK1200)/Term 7 (EK1521)/Telescope Cabinet (EK1501)/Cover2 (EL2042)
//     PlcTask Outputs/GVL_Telescope.close_cover2 <-> Channel 2/GVL_Telescope.close_cover2
//     PlcTask Outputs/GVL_Telescope.open_cover2 <-> Channel 1/GVL_Telescope.open_cover2
//   RoboTelRuntime/RoboTelRuntime Instance <-> Device 1 (EtherCAT)/Term 1 (EK1200)/Term 7 (EK1521)/Telescope Cabinet (EK1501)/Cover3 (EL2042)
//     PlcTask Outputs/GVL_Telescope.close_cover3 <-> Channel 2/GVL_Telescope.close_cover3
//     PlcTask Outputs/GVL_Telescope.open_cover3 <-> Channel 1/GVL_Telescope.open_cover3
//   RoboTelRuntime/RoboTelRuntime Instance <-> Device 1 (EtherCAT)/Term 1 (EK1200)/Term 7 (EK1521)/Telescope Cabinet (EK1501)/Handcontrol IN1 (EL1008)
//     PlcTask Inputs/GVL_pendant_control.BCD1 <-> Channel 1/GVL_pendant_control.BCD1
//     PlcTask Inputs/GVL_pendant_control.BCD2 <-> Channel 2/GVL_pendant_control.BCD2
//     PlcTask Inputs/GVL_pendant_control.BCD4 <-> Channel 3/GVL_pendant_control.BCD4
//     PlcTask Inputs/GVL_pendant_control.BCD8 <-> Channel 4/GVL_pendant_control.BCD8
//     PlcTask Inputs/GVL_pendant_control.direction_down <-> Channel 7/GVL_pendant_control.direction_down
//     PlcTask Inputs/GVL_pendant_control.direction_up <-> Channel 6/GVL_pendant_control.direction_up
//     PlcTask Inputs/GVL_pendant_control.key_switch <-> Channel 8/GVL_pendant_control.key_switch
//     PlcTask Inputs/GVL_pendant_control.reset_switch <-> Channel 5/GVL_pendant_control.reset_switch
//   RoboTelRuntime/RoboTelRuntime Instance <-> Device 1 (EtherCAT)/Term 1 (EK1200)/Term 7 (EK1521)/Telescope Cabinet (EK1501)/Handcontrol IN2 (EL1008)
//     PlcTask Inputs/GVL_pendant_control.direction_left <-> Channel 2/GVL_pendant_control.direction_left
//     PlcTask Inputs/GVL_pendant_control.direction_right <-> Channel 3/GVL_pendant_control.direction_right
//     PlcTask Inputs/GVL_pendant_control.start_switch <-> Channel 1/GVL_pendant_control.start_switch
//   RoboTelRuntime/RoboTelRuntime Instance <-> Device 1 (EtherCAT)/Term 1 (EK1200)/Term 7 (EK1521)/Telescope Cabinet (EK1501)/Handcontrol OUT (EL2008)
//     PlcTask Outputs/GVL_pendant_control.lamp_down <-> Channel 2/GVL_pendant_control.lamp_down
//     PlcTask Outputs/GVL_pendant_control.lamp_error <-> Channel 5/GVL_pendant_control.lamp_error
//     PlcTask Outputs/GVL_pendant_control.lamp_left <-> Channel 4/GVL_pendant_control.lamp_left
//     PlcTask Outputs/GVL_pendant_control.lamp_right <-> Channel 3/GVL_pendant_control.lamp_right
//     PlcTask Outputs/GVL_pendant_control.lamp_up <-> Channel 1/GVL_pendant_control.lamp_up
//   RoboTelRuntime/RoboTelRuntime Instance <-> Device 1 (EtherCAT)/Term 1 (EK1200)/Term 7 (EK1521)/Telescope Cabinet (EK1501)/Hydraulics IN (EL1008)
//     PlcTask Inputs/GVL_Hydraulics.oil_reserve <-> Channel 2/GVL_Hydraulics.oil_reserve
//     PlcTask Inputs/GVL_Hydraulics.oilpan_maximum <-> Channel 1/GVL_Hydraulics.oilpan_maximum
//   RoboTelRuntime/RoboTelRuntime Instance <-> Device 1 (EtherCAT)/Term 1 (EK1200)/Term 7 (EK1521)/Telescope Cabinet (EK1501)/Limits IN1 (EL1008)
//     PlcTask Inputs/GVL_Telescope.focus_limit_far <-> Channel 2/GVL_Telescope.focus_limit_far
//     PlcTask Inputs/GVL_Telescope.focus_limit_near <-> Channel 1/GVL_Telescope.focus_limit_near
//     PlcTask Inputs/GVL_Telescope.nasmyth_limit_left <-> Channel 3/GVL_Telescope.nasmyth_limit_left
//     PlcTask Inputs/GVL_Telescope.nasmyth_limit_right <-> Channel 4/GVL_Telescope.nasmyth_limit_right
//   RoboTelRuntime/RoboTelRuntime Instance <-> Device 1 (EtherCAT)/Term 1 (EK1200)/Term 7 (EK1521)/Telescope Cabinet (EK1501)/M3 (EL2042)
//     PlcTask Outputs/NasmythControl.nasmyth_move_left <-> Channel 2/NasmythControl.nasmyth_move_left
//     PlcTask Outputs/NasmythControl.nasmyth_move_right <-> Channel 1/NasmythControl.nasmyth_move_right
//   RoboTelRuntime/RoboTelRuntime Instance <-> Device 1 (EtherCAT)/Term 1 (EK1200)/Term 7 (EK1521)/Telescope Cabinet (EK1501)/Temp2 (EL3202-0010)
//     PlcTask Inputs/GVL_Telescope.temperature_mirror1 <-> RTD Inputs Channel 2/GVL_Telescope.temperature_mirror1
//     PlcTask Inputs/GVL_Telescope.temperature_mirror2 <-> RTD Inputs Channel 1/GVL_Telescope.temperature_mirror2
//   RoboTelRuntime/RoboTelRuntime Instance <-> Device 1 (EtherCAT)/Term 1 (EK1200)/Term 7 (EK1521)/Telescope Cabinet (EK1501)/Temp4 (EL3202-0010)
//     PlcTask Inputs/GVL_Telescope.temperature_cabinet <-> RTD Inputs Channel 2/GVL_Telescope.temperature_cabinet
//   RoboTelRuntime/RoboTelRuntime Instance <-> Device 1 (EtherCAT)/Term 1 (EK1200)/Term 7 (EK1521)/Weather (EK1501)/Analog IN (EL3068)
//     PlcTask Inputs/GVL_Environment.rawBrightness <-> AI Standard Channel 6/GVL_Environment.rawBrightness
//     PlcTask Inputs/GVL_Environment.rawHumidity <-> AI Standard Channel 4/GVL_Environment.rawHumidity
//     PlcTask Inputs/GVL_Environment.rawLightDirection <-> AI Standard Channel 7/GVL_Environment.rawLightDirection
//     PlcTask Inputs/GVL_Environment.rawPrecipitation <-> AI Standard Channel 8/GVL_Environment.rawPrecipitation
//     PlcTask Inputs/GVL_Environment.rawPressure <-> AI Standard Channel 5/GVL_Environment.rawPressure
//     PlcTask Inputs/GVL_Environment.rawTemperature <-> AI Standard Channel 3/GVL_Environment.rawTemperature
//     PlcTask Inputs/GVL_Environment.rawWindDirection <-> AI Standard Channel 2/GVL_Environment.rawWindDirection
//     PlcTask Inputs/GVL_Environment.rawWindSpeed <-> AI Standard Channel 1/GVL_Environment.rawWindSpeed
//   RoboTelRuntime/RoboTelRuntime Instance <-> Device 1 (EtherCAT)/Term 1 (EK1200)/Term 7 (EK1521)/Weather (EK1501)/Rain IN (EL1008)
//     PlcTask Inputs/GVL_Environment.rawNoRain <-> Channel 1/GVL_Environment.rawNoRain
//     PlcTask Inputs/GVL_Environment.rawRain <-> Channel 2/GVL_Environment.rawRain
//   RoboTelRuntime/RoboTelRuntime Instance <-> Device 1 (EtherCAT)/Term 1 (EK1200)/Term 84 (EK1521)/Filterwheel Cabinet (EK1501)/Filterrad (EL7211-0010)
//     PlcTask Inputs/GVL_FilterWheel.bCalibrationCam <-> FB Touch probe status/Touch probe status/TP1 Input
//   RoboTelRuntime/RoboTelRuntime Instance <-> Device 1 (EtherCAT)/Term 1 (EK1200)/Term 84 (EK1521)/Filterwheel Cabinet (EK1501)/Term 24 (EL3064)
//     PlcTask Inputs/GVL_Auxiliary.pressure_Dewar <-> AI Standard Channel 1/GVL_Auxiliary.pressure_Dewar
//   RoboTelRuntime/RoboTelRuntime Instance <-> Device 1 (EtherCAT)/Term 1 (EK1200)/TwinSAFE Logic (EL6910)
//     PlcTask Inputs/GVL_Safety.Error <-> StandardInputs/TwinSafeGroup1.SafetyError_14
//     PlcTask Outputs/GVL_Safety.ErrAck <-> StandardOutputs/TwinSafeGroup1.ErrorAcknowledgement_1
//     PlcTask Outputs/GVL_Safety.Restart <-> StandardOutputs/TwinSafeGroup1.RestartSafety_13
//     PlcTask Outputs/GVL_Safety.Run <-> StandardOutputs/TwinSafeGroup1.RunSafety_11
//   RoboTelRuntime/RoboTelRuntime Instance <-> NC-Task 1 SAF/Axes/Azimuth
//     PlcTask Inputs/GVL_Telescope.AzimuthAxisRef.NcToPlc <-> Outputs/ToPlc
//     PlcTask Outputs/GVL_Telescope.AzimuthAxisRef.PlcToNc <-> Inputs/FromPlc
//   RoboTelRuntime/RoboTelRuntime Instance <-> NC-Task 1 SAF/Axes/Derotator
//     PlcTask Inputs/GVL_Telescope.DerotatorAxisRef.NcToPlc <-> Outputs/ToPlc
//     PlcTask Outputs/GVL_Telescope.DerotatorAxisRef.PlcToNc <-> Inputs/FromPlc
//   RoboTelRuntime/RoboTelRuntime Instance <-> NC-Task 1 SAF/Axes/DomeAzimuth
//     PlcTask Inputs/GVL_Dome.ActVelo <-> Outputs/ToPlc/ActVelo
//     PlcTask Inputs/GVL_Dome.DomeAxisRef.NcToPlc <-> Outputs/ToPlc
//     PlcTask Inputs/GVL_Dome.bBreak <-> Drive/Outputs/Out/bBreak
//     PlcTask Inputs/GVL_Dome.bDirectionMinus <-> Drive/Outputs/Out/bDirectionMinus
//     PlcTask Inputs/GVL_Dome.bDirectionPlus <-> Drive/Outputs/Out/bDirectionPlus
//     PlcTask Inputs/GVL_Dome.bVeloHigh <-> Drive/Outputs/Out/bVeloHigh
//     PlcTask Inputs/GVL_Dome.bVeloLow <-> Drive/Outputs/Out/bVeloLow
//     PlcTask Outputs/GVL_Dome.DomeAxisRef.PlcToNc <-> Inputs/FromPlc
//   RoboTelRuntime/RoboTelRuntime Instance <-> NC-Task 1 SAF/Axes/Elevation
//     PlcTask Inputs/GVL_Telescope.ElevationAxisRef.NcToPlc <-> Outputs/ToPlc
//     PlcTask Outputs/GVL_Telescope.ElevationAxisRef.PlcToNc <-> Inputs/FromPlc
//   RoboTelRuntime/RoboTelRuntime Instance <-> NC-Task 1 SAF/Axes/Filterrad
//     PlcTask Inputs/GVL_FilterWheel.FilterWheel_AxisRef.NcToPlc <-> Outputs/ToPlc
//     PlcTask Outputs/GVL_FilterWheel.FilterWheel_AxisRef.PlcToNc <-> Inputs/FromPlc
//   RoboTelRuntime/RoboTelRuntime Instance <-> NC-Task 1 SAF/Axes/Focus
//     PlcTask Inputs/GVL_Telescope.FocusAxisRef.NcToPlc <-> Outputs/ToPlc
//     PlcTask Outputs/GVL_Telescope.FocusAxisRef.PlcToNc <-> Inputs/FromPlc

CONFIGURATION RoboTelRuntime
    RESOURCE PLC ON TwinCAT3
        TASK PlcTask(INTERVAL := T#10ms, PRIORITY := 14);
        PROGRAM MAIN WITH PlcTask : MAIN;
    END_RESOURCE
END_CONFIGURATION

// ---- DUTs/E_TCSCommand.TcDUT
{attribute 'qualified_only'}
{attribute 'strict'}
TYPE E_TCSCommand :
(
	no_command := 0,
	gohome,
	park,
	track,
	goto,
	stop,
	pumping,
	slew
);
END_TYPE

// ---- DUTs/E_TCSErrors.TcDUT
{attribute 'qualified_only'}
{attribute 'strict'}
TYPE E_TCSErrors :
(
	no_error := 0,
	info :=1,
	warning := 2,
    error := 4,
	panic := 8
);
END_TYPE

// ---- DUTs/E_TelescopeMode.TcDUT
{attribute 'qualified_only'}
{attribute 'strict'}
TYPE E_TelescopeMode :
(
	off := 0,
	manual := 1,
	automatic := 2
);
END_TYPE

// ---- DUTs/ST_DomeStruct.TcDUT
TYPE ST_DomeStruct :
STRUCT
	OpenShutter: 	BOOL;
	CloseShutter: 	BOOL;
	OpenFlap: 		BOOL;
	CloseFlap: 		BOOL;
	WatchDogReset:	BOOL;
END_STRUCT
END_TYPE

// ---- GVLs/GVL_Auxiliary.TcGVL
{attribute 'qualified_only'}
VAR_GLOBAL
	// Dewar Temperature sensor error
	Dewar_temperature_error	AT%I*: BOOL;
	// dewar pressure 0..10V Pfeiffer 
	pressure_Dewar			AT%I*: INT;
	// dewar raw temperature
	temperature_Dewar 		AT%I*: INT;
	
END_VAR

// ---- GVLs/GVL_Dome.TcGVL
{attribute 'qualified_only'}
VAR_GLOBAL
	// clockwise rotation of the dome azimuth	
	Clockwise				AT%I*:	BOOL;
	// counterclockwise rotation of the dome azimuth	
	CounterClockwise		AT%I*:	BOOL;
	// PLC NC command direction +
	bDirectionMinus 		AT%I*:	BOOL;
	// PLC NC command direction -
	bDirectionPlus 			AT%I*:	BOOL;
	// PLC NC command velocity low
	bVeloLow 				AT%I*:	BOOL;
	// PLC NC command velocity high
	bVeloHigh 				AT%I*:	BOOL;
	// PLC NC command break
	bBreak 					AT%I*:	BOOL;
	//bBreakInv 				AT%I*:	BOOL;
	
	// enable the azimuth inverter
	Inverter_Enable 		AT%Q*:	BOOL;
	// negative direction of the azimuth inverter
	Inverter_DirectionMinus AT%Q*: BOOL;
	Inverter_Velocity 		AT%Q*: UINT;
	// light relais
	Light					AT%Q*: 	BOOL;
	// dehumidifier MOSFET
	DeHumidifier			AT%Q*: 	BOOL;
	// EL5151
	// Azimut_raw				AT%I*:	INT;
	// Azimuth home signal
	Azimuth_home				AT%I*:	BOOL;
	
	ActVelo					AT%I*:	LREAL;
	// stop signal
	//Stop:							BOOL;
	// Dome Axis Reference for the azimuth
	DomeAxisRef: 					AXIS_REF;
	// ControlWord to be read by the dome PLC
	DomeControlWord			AT%MW0:	WORD;
END_VAR

// ---- GVLs/GVL_Environment.TcGVL
{attribute 'qualified_only'}

VAR_GLOBAL
	// Input 1
	rawWindSpeed				AT%I*:	INT;
	// Input 2
	rawWindDirection			AT%I*:	INT;
	// Input 3
	rawTemperature				AT%I*:	INT;
	// Input 4
	rawHumidity					AT%I*:	INT;
	// Input 5
	rawPressure 				AT%I*:	INT;
	// Input 6
	rawBrightness				AT%I*:	INT;
	// Input 7
	rawLightDirection			AT%I*:	INT;
	// Input 8
	rawPrecipitation			AT%I*:	INT;
	// Digital Input 1
	rawNoRain					AT%I*:	BOOL;
	// Digital Input 2
	rawRain						AT%I*:	BOOL;
	
	// indoors
	rawHumidityDome				AT%I*:	INT;
	rawTemperatureDome			AT%I*:	INT;
END_VAR

// ---- GVLs/GVL_FilterWheel.TcGVL
{attribute 'qualified_only'}
VAR_GLOBAL
	FilterWheel_AxisRef:	AXIS_REF;
	bCalibrationCam			AT%I*:	BOOL;
END_VAR

// ---- GVLs/GVL_pendant_control.TcGVL
{attribute 'qualified_only'}
//TODO update to current RoboTel IOs
VAR_GLOBAL
	//DIN17 2.0
	BCD1		AT%I*: BOOL;
	//DIN18 2.1
	BCD2		AT%I*: BOOL;
	//DIN19 2.2
	BCD4		AT%I*: BOOL;
	//DIN20 2.3
	BCD8		AT%I*: BOOL;
	//DIN21 2.4
	reset_switch	AT%I*: BOOL;
	//DIN22 2.5
	direction_up	AT%I*: BOOL;
	//DIN23 2.6
	direction_down	AT%I*: BOOL;
	//DIN24 2.7
	key_switch		AT%I*: BOOL;
	//DIN25 3.0 (enable)
	start_switch	AT%I*: BOOL;
	//DIN26 3.1
	direction_left	AT%I*: BOOL;
	//DIN27 3.2
	direction_right	AT%I*: BOOL;
	
	// Outputs
	
	//DOUT9 1.0
	lamp_up			AT%Q*: BOOL;
	//DOUT10 1.1
	lamp_down			AT%Q*: BOOL;
	//DOUT11 1.2
	lamp_right			AT%Q*: BOOL;
	//DOUT12 1.3
	lamp_left			AT%Q*: BOOL;
	//DOUT13 1.4
	lamp_error			AT%Q*: BOOL;
	
END_VAR

// ---- GVLs/GVL_Hydraulics.TcGVL
{attribute 'qualified_only'}
VAR_GLOBAL
	// 2.1
	oil_low				AT%I*: BOOL;
	// ?
	oil_high			AT%I*: BOOL;
	// 2.3
	oil_pressure_OK		AT%I*: BOOL;
	// 2.4
	oil_overtemperature		AT%I*: BOOL;
	// 2.5
	oil_undertemperature	AT%I*: BOOL;
	// 2.6
	oilfilter_dirty		AT%I*: BOOL;
	// 2.7
	pump_running		AT%I*: BOOL;
	// 2.8
	suction_running		AT%I*: BOOL;
	//BT2
	//oil_temperature			AT%I*: INT;
	
	//DIN39 4.6
	oilpan_maximum		AT%I*: BOOL;
	//DIN40 4.7
	oil_reserve			AT%I*: BOOL;
	
		
	//DOUT4 0.3
	oil_pump_enable		AT%Q*: BOOL;
	//DOUT5 0.4
	oil_suction_enable		AT%Q*: BOOL;	
END_VAR

// ---- GVLs/GVL_Safety.TcGVL
{attribute 'qualified_only'}
VAR_GLOBAL
	// Safety Error Condition
	Error		AT%I*:BOOL;
	// Run/Stop Safety
	Run			AT%Q*:BOOL;
	// Restart Safety
	Restart		AT%Q*:BOOL;
	// Error Acknowledgement 
	ErrAck		AT%Q*:BOOL;
END_VAR

// ---- GVLs/GVL_Telescope.TcGVL
{attribute 'qualified_only'}
VAR_GLOBAL
	// BT9 mirror
	temperature_mirror2		AT%I*: INT;
	// BT10
	temperature_mirror1		AT%I*: INT;
	// BT15
	temperature_cabinet		AT%I*: INT;

	//DOUT6 0.5
	brake_azimuth_eve	AT%Q*: BOOL;
	
	// DIN28 3.3 (absolute)
	azimut_limit_switch	AT%I*: BOOL;
	// DIN29 3.4
	focus_limit_near	AT%I*: BOOL;
	// DIN30 3.5
	focus_limit_far		AT%I*: BOOL;
	// DIN31 3.6
	nasmyth_limit_left	AT%I*: BOOL;
	// DIN32 3.7
	nasmyth_limit_right	AT%I*: BOOL;
	
	// DIN35 4.2
	cover2_open		AT%I*: BOOL;
	// DIN36 4.3
	cover2_closed	AT%I*: BOOL;
	// DIN37 4.4
	cover3_open		AT%I*: BOOL;
	// DIN38 4.5
	cover3_closed	AT%I*: BOOL;

	open_cover2		AT%Q*: BOOL;
	close_cover2	AT%Q*: BOOL;
	open_cover3		AT%Q*: BOOL;
	close_cover3	AT%Q*: BOOL;
	
	//DOUT14 1.5
	focus_unlock		AT%Q*: BOOL;
	//DOUT15 4.6
	nasmyth_lock	AT%Q*: BOOL;
	//Horn 4.7
	horn			AT%Q*: BOOL;
	
	// digitale inputs der Endlagen
	Derotator_inputs		AT%I*: WORD;
	// derotator torque feedback
	Derotator_torque		AT%I*: INT;
	
	// digital inputs for limit switches
	Elevation_inputs		AT%I*: WORD;
	// diagnostic number
	Elevation_diagnostic	AT%I*: UDINT;
	// torque feedback
	Elevation_torque		AT%I*: INT;
	
	// digital inputs for limit switches
	Azimuth_inputs			AT%I*: WORD;
	// diagnostic number
	Azimuth_diagnostic		AT%I*: UDINT;
	// torque feedback
	Azimuth_torque			AT%I*: INT;
	
	// Zyklisches Interface zwischen NC und Achse
	AzimuthAxisRef: 	AXIS_REF;
	ElevationAxisRef: 	AXIS_REF;
	DerotatorAxisRef: 	AXIS_REF;
 	// Motor1 Channel 1
	FocusAxisRef:		AXIS_REF;
	
END_VAR

// ---- GVLs/GVL_Main.TcGVL
{attribute 'qualified_only'}
//TODO update to current RoboTel IOs
VAR_GLOBAL
	//DIN1 0.0
	phase_available		AT%I*: BOOL;
	power_available		AT%I*: BOOL;
	L1_L2_Voltage		AT%I*: REAL;
	L2_L3_Voltage		AT%I*: REAL;
	L3_L1_Voltage		AT%I*: REAL;
	//DIN2 0.1
	//key_switch			AT%I*: BOOL;
	//DIN3 0.2
	key_switch_remote	AT%I*: BOOL;
	//DIN4 0.3
	start_switch		AT%I*: BOOL;
	//DIN5 0.4
	stop_switch			AT%I*: BOOL;
	//DIN8 0.7
	reset_switch		AT%I*: BOOL;
	
	//BT1
	main_cabinet_temperature	AT%I*: INT;
	//DIN15 1.6
	brake_clearing		AT%I*: BOOL;
	
	//DOUT1 0.0
	lamp_power			AT%Q*: BOOL;
	//DOUT2 0.1
	lamp_ready			AT%Q*: BOOL;
	//DOUT3 0.2
	lamp_error			AT%Q*: BOOL;
	
	//DOUT7 0.6
	softstart_trafo		AT%Q*:BOOL;

	isRoboTel:		BOOL;
END_VAR

// ---- POUs/MAIN.TcPOU
PROGRAM MAIN
VAR
	// indicates the phases for the hydraulics
	phase_available:	BOOL;
	// telescope drives are ready to enable
	ready:				BOOL;
	// error stat on drive, power or hydraulics
	error:				BOOL;
	// manual, panel or remote reset
	reset:				BOOL;
	// reset from API
	remote_reset:			BOOL;
	// hydraulics warning 
	warning:			BOOL;
	// start hydraulics
	start:				BOOL;
	// start from API
	remote_start:		BOOL;
	// stop hydraulics 
	stop:				BOOL;
	// stop from API
	remote_stop:		BOOL;
	// soft start trafo
	key_switch:			BOOL;
	//	open brake
	brake_clearing:		BOOL := FALSE;
	// blink error lamp on warning
	warn_blink: 		FB_BLINK;
	// main cabinet temperature in degrees
	cabinet_temperature:	REAL;
	ups_output_voltage:		REAL;
	ups_output_current:		REAL;
	ups_output_power:		REAL;
	
	PhaseLog:				FB_EventLog;
	TemperatureEvent:		FB_EventLog;
	UPSEvent:				FB_EventLog;
	
	MQTTTimer : 		TON := (PT:=T#5S);
	GetHostName:		FB_GetHostName;
	HostName: 			STRING(255);
	LightSwitch:		FB_ButtonEnable;
	Lightbutton: 		BOOL;
	bExecute:			BOOL := TRUE;
	cabinet_temperature_warning:	SR;
	
	MQTTClient:		FB_MQTTCommunication;
	
	UPS:		PS_Q4_DcUpsEC_Cyclic_2;
	arrInputPD AT%I*:	ARRAY [0..30] OF WORD;
END_VAR

(* 
Main control loop
* Execute sub modules
* power management
* control panel switches and status lamps

* start switch activates Hydraulics and Trafo
* 
*)
GetHostName(bExecute := bExecute, sHostName => HostName);
bExecute := FALSE;
GVL_Main.isRoboTel := HostName = 'CX-4E6032';
start := GVL_Main.start_switch OR remote_start;
stop := GVL_Main.stop_switch OR remote_stop;

phase_available := GVL_Main.L1_L2_Voltage > 380.0 AND  GVL_Main.L2_L3_Voltage > 380.0 AND  GVL_Main.L3_L1_Voltage > 380.0;
reset := GVL_Main.reset_switch OR GVL_pendant_control.reset_switch OR remote_reset;		
key_switch := GVL_Main.key_switch_remote;
brake_clearing := GVL_Main.brake_clearing;
cabinet_temperature := INT_TO_REAL(GVL_Main.main_cabinet_temperature) / 100.0;
cabinet_temperature_warning(SET1 := cabinet_temperature > 40.0,
							RESET := cabinet_temperature < 35.0);

IF start THEN
	HydraulicsControl.start := TRUE;
	// SimpleLog(Message := 'manual Hydraulics start');
END_IF
IF stop THEN
	HydraulicsControl.stop := TRUE;
	// SimpleLog(Message := 'manual Hydraulics stop');
END_IF

// telescope is ready when power available and hydraulics ok
ready := Transformer.power_OK AND HydraulicsControl.oil_pressure_OK;
		
TelescopeControl();	//
DomeControl();	//
CoverControl();	//
PendantControl();	//
NasmythControl();	//
HydraulicsControl();	//
// deactivate noisy fan if we are on manual
FanControl(enable := NOT PendantControl.manual);
ElevationControl();	//
AzimuthElevationControl();	//
DerotatorControl();	//
FilterWheelControl();	//
FocusControl();
Environment();	//
AuxiliaryControl(); //
MQTTClient();
Transformer();

IF key_switch THEN
	Transformer.start();
ELSE
	Transformer.stop();
END_IF

IF reset THEN
	Transformer.reset();
END_IF

warn_blink(ENABLE := HydraulicsControl.oil_warning OR HydraulicsControl.oil_hot, 
	Q => warning);
error := Transformer.error OR 
			HydraulicsControl.pressure_failure 
			OR (NOT phase_available)
			OR GVL_Telescope.azimut_limit_switch
			//OR PendantControl.error
			OR FanControl.error
			OR ElevationControl.error
			OR FilterWheelControl.Error
			OR DomeControl.Error
			OR Focuscontrol.Error
			OR NasmythControl.error
			OR CoverControl.Error
			OR AzimuthElevationControl.error
			OR DerotatorControl.Error
			OR GVL_Safety.Error;
// set control lights					
GVL_Main.lamp_ready := ready;
GVL_Main.lamp_error := error OR warning;
GVL_Main.lamp_power := Transformer.power_ok AND phase_available;
SafetyHandling();

// UPS Handling
UPS(xActivate := key_switch, 
	arrInputPD := arrInputPD);
	

ups_output_voltage 		:= UPS.wOutputVoltage / 1000.0;
ups_output_current 		:= UPS.wOutputCurrent / 1000.0;
ups_output_power		:= ups_output_voltage * ups_output_current;

LightSwitch(SET := Lightbutton, Q := DomeControl.Light);

MQTTTimer(IN:=TRUE);
IF MQTTTimer.Q THEN // publish new payload every second
	MQTTTimer(IN:=FALSE);
	MQTTClient.Publish('electronics', 'base', 'MainCabinetTemperature', LREAL_TO_FMTSTR(cabinet_temperature, 2, TRUE));
	MQTTClient.Publish('electronics', 'base', 'PowerOK', BOOL_TO_STRING(Transformer.power_ok));
	MQTTClient.Publish('electronics', 'base', 'PhaseOK', BOOL_TO_STRING(phase_available));
	MQTTClient.Publish('electronics', 'base', 'MainReady', BOOL_TO_STRING(ready));
	MQTTClient.Publish('electronics', 'base', 'MasterError', BOOL_TO_STRING(error));
	MQTTClient.Publish('electronics', 'base', 'UPSOutputVoltage', LREAL_TO_FMTSTR(ups_output_voltage, 3, TRUE));
	MQTTClient.Publish('electronics', 'base', 'UPSOutputCurrent', LREAL_TO_FMTSTR(ups_output_current, 3, TRUE));
	MQTTClient.Publish('electronics', 'base', 'UPSOutputPower', LREAL_TO_FMTSTR(ups_output_power, 3, TRUE));
END_IF

PhaseLog(	
	Trigger := 		NOT phase_available, 
	Level := 		ADSLOG_MSGTYPE_ERROR,
	FormatString :=	'%s',
	OnMessage := 	'electrical phases:	ERROR!',
	OffLevel := 	ADSLOG_MSGTYPE_HINT,
	OffMEssage := 	'electrical phases:	active');

TemperatureEvent(	
	Trigger := 		cabinet_temperature_warning.Q1, 
	Level := 		ADSLOG_MSGTYPE_WARN,
	FormatString :=	'Main Cabinet Temperature warning:	%s',
	OnMessage := 	LREAL_TO_FMTSTR( cabinet_temperature, 1, TRUE),);
	
UPSEvent(	
	Trigger := 		UPS.xAlarm, 
	Level := 		ADSLOG_MSGTYPE_ERROR,
	FormatString :=	'%s',
	OnMessage := 	'UPS Alarm!');

END_PROGRAM

// ---- POUs/FunctionBlocks/FB_BLINK.TcPOU
FUNCTION_BLOCK FB_BLINK
VAR_INPUT
	ENABLE:		BOOL;
	ON_TIME:	TIME := T#500MS;
	OFF_TIME:	TIME := T#500MS;
END_VAR
VAR_OUTPUT
	Q:		BOOL;
END_VAR
VAR
    IMPULS   :TOF;
    PAUSE    :TOF;
END_VAR

IMPULS(IN:= NOT PAUSE.Q AND NOT IMPULS.Q, PT:= ON_TIME);
PAUSE(IN:= NOT PAUSE.Q AND NOT IMPULS.Q, PT:= OFF_TIME);
Q := IMPULS.Q AND ENABLE;

END_FUNCTION_BLOCK

// ---- POUs/FunctionBlocks/FB_EventLog.TcPOU
FUNCTION_BLOCK FB_EventLog
VAR_INPUT
	Trigger:		BOOL;
	// ADSLOG_MSGTYPE_HINT or ADSLOG_MSGTYPE_WARN or ADSLOG_MSGTYPE_ERROR
	Level:			UDINT := ADSLOG_MSGTYPE_HINT;
	FormatString: 	STRING(255) := '%s';
	OnMessage: 		STRING(255) := '';
	OffMessage:		STRING(255) := '';
	OffLevel:		UDINT := ADSLOG_MSGTYPE_HINT;
END_VAR
VAR_OUTPUT
END_VAR
VAR
	LogonTrigger: R_TRIG;
	LogoffTrigger: F_TRIG; // R_Trig or F_Trig ?!
	PayloadMessage: STRING(255);
	fbFormat:	FB_FormatString;
	LevelString: STRING;
END_VAR

LogonTrigger(CLK := Trigger);
LogoffTrigger(CLK := Trigger);
// in case the OffLevel is not set use the default Level Value
IF OffLevel = 0 THEN
	OffLevel := Level;
END_IF
IF LogonTrigger.Q AND LEN(OnMessage)>0 THEN
	ADSLOGSTR( Level OR ADSLOG_MSGTYPE_LOG, FormatString, OnMessage);
END_IF

IF LogoffTrigger.Q AND LEN(OffMessage)>0 THEN
	ADSLOGSTR( OffLevel OR ADSLOG_MSGTYPE_LOG, FormatString, OffMessage);
END_IF

IF LogonTrigger.Q AND LEN(OnMessage)>1 THEN
	IF Level=ADSLOG_MSGTYPE_HINT THEN
		LevelString := 'INFO';
	ELSIF Level=ADSLOG_MSGTYPE_WARN THEN
		LevelString := 'WARNING';
	ELSE
	    LevelString := 'ERROR';
	END_IF
	fbFormat( sFormat := FormatString, arg1 := F_STRING(OnMessage), sOut => PayloadMessage);
	MAIN.MQTTClient.PublishLog(LevelString, PayloadMessage);

END_IF

IF LogoffTrigger.Q AND LEN(OffMessage)>1 THEN
	IF OffLevel=ADSLOG_MSGTYPE_HINT THEN
		LevelString := 'INFO';
	ELSIF OffLevel=ADSLOG_MSGTYPE_WARN THEN
		LevelString := 'WARNING';
	ELSE
	    LevelString := 'ERROR';
	END_IF
	fbFormat( sFormat := FormatString, arg1 := F_STRING(OffMessage), sOut => PayloadMessage);
	MAIN.MQTTClient.PublishLog(LevelString, PayloadMessage);
END_IF

END_FUNCTION_BLOCK

// ---- POUs/Functions/Trigger.TcPOU
FUNCTION Trigger : BOOL
VAR_INPUT
	// Trigger is TRUE if Signal changes state
	Signal:	BOOL;
END_VAR
VAR
	fsignal:	F_TRIG;
	rsignal:	R_TRIG;
END_VAR

fsignal(CLK := Signal);
rsignal(CLK := Signal);

Trigger := fsignal.Q OR rsignal.Q;

END_FUNCTION

// ---- POUs/FunctionBlocks/FB_ButtonEnable.TcPOU
FUNCTION_BLOCK FB_ButtonEnable
VAR_INPUT
	SET:	BOOL;
	RESET:	BOOL;
END_VAR
VAR_IN_OUT
	Q: BOOL;
END_VAR
VAR
	trigger:	R_TRIG;
//	ftrigger:	F_TRIG;
END_VAR

trigger(CLK := SET);
//ftrigger(CLK := SET);

// if button was triggered, flip the state of the output
IF trigger.Q THEN
	Q := NOT Q;
END_IF

// if reset is enabled we disable the output
IF RESET THEN
	Q := FALSE;
END_IF

END_FUNCTION_BLOCK

// ---- POUs/FunctionBlocks/FB_MQTTCommunication.TcPOU
FUNCTION_BLOCK FB_MQTTCommunication
VAR_INPUT
END_VAR
VAR_OUTPUT
END_VAR
VAR
	GetHostName:		FB_GetHostName;
	HostName: 			STRING(255);
    bSetParameter:		BOOL := FALSE;
    bConnect:			BOOL := FALSE;
    (* received message *)
	bSubscribed: 		BOOL;
	sTopicSub: 			STRING(255) := 'RoboTel/Telescope/SET';
	{attribute 'TcEncoding':='UTF-8'}
	sTopicRcv: 			STRING(255);
	{attribute 'TcEncoding':='UTF-8'}
	fbMessageQueue:		FB_IotMqttMessageQueue;
    fbMessage:			FB_IotMqttMessage;
	fbMqttClient:		FB_IotMqttClient;
	sPayloadRcv: 		STRING;
	influxMessage:		FB_InfluxMessage;
	measurement, 
	parameter, 
	value:		STRING(255);
END_VAR

(*
MQTT Communication section

Source:
https://infosys.beckhoff.com/english.php?content=../content/1033/tf6701_tc3_iot_communication_mqtt/3518541195.html&id=

*)
IF HostName='' THEN
	GetHostName.bExecute := TRUE;
ELSE
	GetHostName.bExecute := FALSE;
	bSetParameter := TRUE;
END_IF

GetHostName(sHostName => HostName);

// set the parameters once
IF bSetParameter THEN
    bSetParameter               := FALSE;
    fbMqttClient.sHostName      := 'primitivo.aip.de';
    fbMqttClient.nHostPort      := 1883;
    fbMqttClient.sClientId      := HostName; 
    fbMqttClient.sTopicPrefix   := ''; 
	fbMqttClient.nKeepAlive     := 60; 
    fbMqttClient.ipMessageQueue := fbMessageQueue;
	bConnect := TRUE;
END_IF

// connect to the client
IF NOT fbMqttClient.bConnected THEN
;
END_IF

fbMqttClient.Execute(bConnect);
	
IF fbMqttClient.bConnected THEN
    IF NOT bSubscribed THEN
        bSubscribed := fbMqttClient.Subscribe(sTopic:=sTopicSub, 
												eQoS:=TcIotMqttQos.AtMostOnceDelivery);
    END_IF
END_IF

// receive queued messages
IF fbMessageQueue.nQueuedMessages > 0 THEN
    IF fbMessageQueue.Dequeue(fbMessage:=fbMessage) THEN
        fbMessage.GetTopic(pTopic:=ADR(sTopicRcv), nTopicSize:=SIZEOF(sTopicRcv) );
        fbMessage.GetPayload(pPayload:=ADR(sPayloadRcv), nPayloadSize:=SIZEOF(sPayloadRcv), bSetNullTermination:=TRUE);
		ADSLOGSTR( ADSLOG_MSGTYPE_HINT OR ADSLOG_MSGTYPE_LOG, 'MQTT %s', sPayloadRcv);
		IF sTopicRcv = sTopicSub THEN
			influxMessage(  sPayload := sPayloadRcv, measurement => measurement, parameter => parameter, value => value);
			IF measurement = 'command' THEN
				IF parameter = 'power' THEN
					TelescopeControl.power := STRING_TO_BOOL(value);
				ELSIF parameter = 'park' THEN
					TelescopeControl.park := STRING_TO_BOOL(value);
				ELSIF parameter = 'gohome' THEN
					TelescopeControl.gohome := STRING_TO_BOOL(value);
				ELSIF parameter = 'track' THEN
					TelescopeControl.track := STRING_TO_BOOL(value);
				ELSIF parameter = 'goto' THEN
					TelescopeControl.goto := STRING_TO_BOOL(value);
				ELSIF parameter = 'slew' THEN
					TelescopeControl.slew := STRING_TO_BOOL(value);
				ELSIF parameter = 'stop' THEN
					TelescopeControl.stop := STRING_TO_BOOL(value);
				ELSIF parameter = 'reset' THEN
					TelescopeControl.reset := STRING_TO_BOOL(value);
				ELSIF parameter = 'nasmyth' THEN
					TelescopeControl.Nasmyth_port := STRING_TO_USINT(value);
				ELSIF parameter = 'rightascension' THEN
					TelescopeControl.rightascension := STRING_TO_LREAL(value);
				ELSIF parameter = 'declination' THEN
					TelescopeControl.declination := STRING_TO_LREAL(value);
				ELSIF parameter = 'elevation' THEN
					TelescopeControl.elevation := STRING_TO_LREAL(value);
				ELSIF parameter = 'azimuth' THEN
					TelescopeControl.azimuth := STRING_TO_LREAL(value);
				ELSIF parameter = 'focus' THEN
					TelescopeControl.focus_position := STRING_TO_LREAL(value);
				ELSIF parameter = 'derotator' THEN
					TelescopeControl.derotator_offset := STRING_TO_LREAL(value);
				ELSIF parameter = 'elevationoffset' THEN
					TelescopeControl.elevation_offset := STRING_TO_LREAL(value);
				ELSIF parameter = 'azimuthoffset' THEN
					TelescopeControl.azimuth_offset := STRING_TO_LREAL(value);
				ELSIF parameter = 'derotatoroffset' THEN
					TelescopeControl.derotator_offset := STRING_TO_LREAL(value);ELSE
					ADSLOGSTR( ADSLOG_MSGTYPE_WARN OR ADSLOG_MSGTYPE_LOG, 'MQTT not understood %s', sPayloadRcv);
				END_IF
			END_IF // measurement
		END_IF // Topic
		sPayloadRcv := '';
    END_IF // Dequeue
END_IF

PROPERTY Error : BOOL
GET
Error := fbMqttClient.bError;
END_GET
END_PROPERTY

METHOD Publish : BOOL
VAR_INPUT
	domain: 	STRING(255) := 'environment';
	location: 	STRING(255) := 'roof';
	parameter:	STRING(255);
	value:		STRING(255);
END_VAR
VAR
	sPayloadPub: STRING(255) := '';
	fbFormat:	FB_FormatString;
	bError:		BOOL;
	nErrID: UDINT;
	retain_message:		BOOL := FALSE;
END_VAR
//sPayloadPub := 'environment,location=roof,host=CX-4E6032 ';
fbFormat( sFormat := '%s,location=%s,host=%s %s=%s', 
			arg1 := F_STRING(domain), 
			arg2 := F_STRING(location), 
			arg3 := F_STRING(HostName),
			arg4 := F_STRING(parameter),
			arg5 := F_STRING(value),
 
			sOut => sPayloadPub,
			bError => bError, 
			nErrID => nErrID );
// retain message if value is boolean
retain_message := value = 'TRUE' OR value = 'FALSE';

Publish := fbMqttClient.Publish(	
				sTopic:= 'RoboTel/Telemetry', 
				pPayload:= ADR(sPayloadPub), 
				nPayloadSize:= LEN2(ADR(sPayloadPub)),
				eQoS:= TcIotMqttQos.AtMostOnceDelivery,
				bRetain:= retain_message, 
				bQueue:= FALSE );
END_METHOD

METHOD PublishLog : BOOL
VAR_INPUT
	level: 	STRING(255) := 'INFO';
	message:	STRING(255);
	
END_VAR
VAR
	sPayloadPub: STRING(255) := '';
	fbFormat:	FB_FormatString;
	bError:		BOOL;
	nErrID: UDINT;
END_VAR
VAR_OUTPUT
	published: BOOL;
END_VAR
//sPayloadPub := 'environment,location=roof,host=CX-4E6032 ';
fbFormat( sFormat := 'log,host=%s,level=%s message="%s"', 
			arg1 := F_STRING(HostName), 
			arg2 := F_STRING(level), 
			arg3 := F_STRING(message),
 
			sOut => sPayloadPub,
			bError => bError, 
			nErrID => nErrID );

published := fbMqttClient.Publish(	
				sTopic:= 'RoboTel/Log', 
				pPayload:= ADR(sPayloadPub), 
				nPayloadSize:= LEN2(ADR(sPayloadPub)),
				eQoS:= TcIotMqttQos.AtMostOnceDelivery,
				bRetain:= FALSE, 
				bQueue:= FALSE );
END_METHOD

END_FUNCTION_BLOCK

// ---- POUs/FunctionBlocks/FB_InfluxMessage.TcPOU
FUNCTION_BLOCK FB_InfluxMessage
VAR_INPUT
	// payload string received
	sPayload:	STRING(255);
END_VAR
VAR_OUTPUT
	// measurement string (first word)
	measurement:	STRING(255) := '';
	// parameter (variable name)
	parameter:		STRING(255) := '';
	// value (variable content)
	value:			STRING(255) := '';
END_VAR
VAR
	//space_position:		INT;
	//equial_position:	INT;
	comma_position:		INT;
	measurement_tags:	STRING(255);
	parameter_value: 	STRING(255);
	bResultSplit: 		BOOL;
	// definition of the space separator
	spaceSeparator:		STRING(1) := ' ';
	// definition of the comma separator
	commaSeparator:		STRING(1) := ',';
	// definition of the equial sign separator
	equialSeparator:	STRING(1) := '=';
END_VAR

(* 
parse message in influx format:
	measurement parameter=value
	measurement,tag1=tag1value parameter=value
	TODO:
	measurement,tag1=tag1value parameter1=value1,parameter2=value2

Multiple parameter/value pairs are ignored for now.
tags are not supported.
*)

//separate measurement from parameter, value
bResultSplit := FindAndSplit( pSeparator     := ADR(spaceSeparator), pSrcString := ADR(sPayload), 
                              pLeftString    := ADR(measurement_tags), nLeftSize  := SIZEOF(measurement_tags), 
                              pRightString   := ADR(parameter_value), nRightSize := SIZEOF(parameter_value),
                              bSearchFromRight := FALSE );
IF NOT bResultSplit THEN
	RETURN;
END_IF
// look for tags attached to the measurement
comma_position := FIND(measurement_tags, commaSeparator);
IF comma_position = 0 THEN
	measurement := measurement_tags;
ELSE
	measurement := LEFT(measurement_tags, comma_position-1);
END_IF
// dissect the parameter=value part
comma_position := FIND(parameter_value, commaSeparator);
IF comma_position = 0 THEN
	// we have only one parameter value pair
	bResultSplit := FindAndSplit( pSeparator     := ADR(equialSeparator), pSrcString := ADR(parameter_value), 
                              pLeftString    := ADR(parameter), nLeftSize  := SIZEOF(parameter), 
                              pRightString   := ADR(value), nRightSize := SIZEOF(value),
                              bSearchFromRight := FALSE );

ELSE
	// we have more than one parameter value pair
	parameter_value := LEFT(parameter_value, comma_position-1);
	bResultSplit := FindAndSplit( pSeparator     := ADR(equialSeparator), pSrcString := ADR(parameter_value), 
                              pLeftString    := ADR(parameter), nLeftSize  := SIZEOF(parameter), 
                              pRightString   := ADR(value), nRightSize := SIZEOF(value),
                              bSearchFromRight := FALSE );
	// TODO: return the rest an re-parse
END_IF

END_FUNCTION_BLOCK

// ---- POUs/TelescopeControl.TcPOU
PROGRAM TelescopeControl
VAR_INPUT
(*
TCS interface section
see https://gitlab.aip.de/bmk10k/telescope_firmware/snippets/5
*)
	
	// boolean, true: Power on, false: power off
	power: 		BOOL;
	// boolean, true: go to home position, unset track/goto if active
	gohome: 	BOOL;
	// boolean, true: go into park position, ready to stow telescope, unset track/goto
	park: 		BOOL;
	// boolean, TRUE: MOVE telescope TO last ra/de AND start tracking. Set 'goto' TO FALSE, IF TRUE. FALSE: Stop tracking as soon as possible
	track: 		BOOL;
	// boolean, TRUE: MOVE telescope TO tau/de AND stop there. Set track TO FALSE, IF TRUE. FALSE: no effect.)
	goto:		BOOL;	
	// move the telescope to a given az-alt position
	slew:		BOOL;
	// boolean, TRUE: Stop motion OF telescope immediately, set goto AND track TO FALSE. FALSE: Allow motion OF telescope again via track/goto).
	stop:		BOOL;	
	// internal command: telescope is moved to pumping position
	pumping:	BOOL;
	// initiates hard-reset on all axis
	reset:		BOOL;
	// apparent right ascension, degrees, double
	rightascension:			LREAL := (00.0 + 08.0/60.0 + 23.17/3600.0) *15.0;	
	// apparent declination, degrees, double
	declination: 		LREAL := 29.0 + 05.0/60.0 + 26.99/3600.0;
	// desired elevation of the telescope pointing 
	elevation:	LREAL := 45.0;
	// desired azimut of the telescope pointing 
	azimuth:	LREAL := 320.0;
	// absolute offset for elevation
	elevation_offset:	LREAL := 0.0;
	// absolute offset for azimuth
	azimuth_offset : 	LREAL := 0.0;
	// absolute offset for time
	time_offset: 		LREAL := 0.0;
	// offset for the de-rotator
	derotator_offset:	LREAL := 180.0;
	// Nasmyth port 1 or 2
	Nasmyth_port: USINT;
	// Focus position in mm
	focus_position: LREAL := 77.000;
END_VAR
VAR
	// manual or automatic operation of the telescope
	telescope_mode : E_TelescopeMode;	
	// actual command from the TCS
	TCS_command: 	E_TCSCommand;
	// current Julian Date calculated from system time
	jd:	LREAL;
	// image derotation
	derotation_calc:	LREAL;
	// local siderial time calculated from Julian date
	lst:	LREAL;
	// values calulated when ra and dec are set by TCS
	elevation_calc:	LREAL; 
	azimuth_calc:	LREAL;
	// values calulated when azimuth and elevation are set by TCS
	rightascension_calc:	LREAL;
	declination_calc:	LREAL;
	
	
	(* Hour Angle part *)
	Hourangle_calc: LREAL;
	
	fbTime: FB_AstroClock;
	
	eq2hor2:	FB_EQ2HOR2;
	hor2eq:		FB_HOR2EQ;
	sunpos:		FB_SUNPOS;
	sunhor2:	FB_EQ2HOR2;
	// zenith distance of the sun
	solz: 		LREAL;
	// triggers power-failure event
	powerfailure: 	BOOL;
	powerontrigger:		R_TRIG;
	powerofftrigger:		F_TRIG;
	poweronwarning:	TP;
	poweron_reset:	TP;
	power_timeout:	TON;
	
	
	TCSpowerEvent,
	TCSgohomeEvent,
	TCSparkEvent,
	TCSgotoEvent,
	TCStrackEvent,
	TCSstopEvent,
	AltitudeEvent,
	TCSreadyEvent: FB_Eventlog;
	FocusDelay: TON := (PT:=T#5S);
	MQTTTimer : TON := (PT:=T#5S);
	// rotational velocity of the derotator
	DerotatorVelocity: LREAL;
	
	StatusWord, LastStatus:	UDINT;
END_VAR
VAR_OUTPUT
	//		TRUE, IF telescope can be operated
	ready:	BOOL; 
	// indicates an error on one of the components
	error:	BOOL;	
	//error id of axis
	errorid:	UDINT;	
	//TRUE, IF telescope is in fast-MOVE phase (includes pole-swap)
	sliding: BOOL;	
	//TRUE, IF telescope is on tracking position AND currently tracking.
	tracking: BOOL;	
	//TRUE, IF telescope is AT rest.
	stopped: BOOL;	
	// Current tau/dec. in degrees.
	//decurrent, taucurrent: LREAL; 
	// (all degrees, azimuth 0=S, W>0)
	//racurrent: LREAL; 
	elevation_current:	LREAL;
	azimuth_current:	LREAL;
	//	(time in sec. to reach the goto/track position)
	slewtime: LREAL; 
	// 	(TIME in sec. available UNTIL pole-swap necessary).
	//tracktime: LREAL;	
	// True: telescope is calibrated
	homed: BOOL;
END_VAR
VAR CONSTANT
(* Potsdam:
	longitude: LREAL := 13.104589;
	latitude: LREAL := 52.404977;
*)
(* RoboTel site : *)
	// telescope site longitude, source: Google 
	longitude: LREAL := 13.101867;
	// telescope site latitude, source: Google
	latitude: LREAL := 52.404940;
	// telescope site height above sea level: estimated
	altitude: LREAL := 33.0;
	//siderial_velocity: LREAL := 360.0 / 86164.099;
	//position_velocity: LREAL := 1.0;
	elevation_park: LREAL := 70.0;
	azimuth_park: LREAL := 359.999;

	elevation_home: LREAL := 45.0;
	azimuth_home: LREAL := 180.0;
END_VAR

TelescopeAuxiliary();

// get the system time
fbTime();
jd := DateTime2JD(fbTime.time_RTCEX2);
lst := CT2LST(longitude, jd);
// set reset state either by hardware (key pressed) or by software (set by e.g. tcs)
IF GVL_Main.reset_switch THEN
	reset := TRUE;
END_IF


IF ElevationControl.error THEN
	errorid := ElevationControl.ErrorID;
	ElevationControl.reset := reset;
ELSIF AzimuthElevationControl.error THEN
	errorid := AzimuthElevationControl.ErrorID;
	AzimuthElevationControl.Reset := reset;
ELSIF FilterWheelControl.Error THEN
	errorid := FilterWheelControl.ErrorID;
	FilterWheelControl.Reset := reset;
ELSIF DomeControl.Error THEN
	errorid := DomeControl.ErrorID;
	DomeControl.Reset := reset;
ELSIF Focuscontrol.Error THEN
	errorid := Focuscontrol.ErrorID;
	FocusControl.reset := reset;
ELSIF DerotatorControl.Error THEN
	errorid := DerotatorControl.ErrorID;
	DerotatorControl.reset := reset;
END_IF

error := ElevationControl.error OR 
		 AzimuthElevationControl.error OR
		 FilterWheelControl.Error OR
		 // DomeControl.Error OR
		 Focuscontrol.Error OR
		 DerotatorControl.Error;

slewtime := MAX(MAX(ElevationControl.slewtime, AzimuthElevationControl.slewtime), DerotatorControl.slewtime);
			
IF error THEN
	gohome := 	FALSE;
	park  := 	FALSE;
	track := 	FALSE;
	goto := 	FALSE;
	slew := 	FALSE;
	pumping :=	FALSE;
END_IF
		 
IF ElevationControl.error THEN
	ElevationControl.enable := FALSE;
	AzimuthElevationControl.enable := FALSE;
	HydraulicsControl.close_brake := TRUE;
	power := FALSE;
END_IF

(*
IF AzimuthElevationControl.error THEN
	AzimuthElevationControl.enable := FALSE;
END_IF
*)

// determine the operation of the telescope based on the switch set
IF GVL_pendant_control.key_switch THEN
	telescope_mode := E_TelescopeMode.manual;
ELSE
	telescope_mode := E_TelescopeMode.automatic;
END_IF

eq2hor2(alpha := rightascension,
	delta := declination,
	lon := longitude,
	lat := latitude,
	JD := jd + time_offset,
	alt => elevation_calc,
	az => azimuth_calc,
	ha => hourangle_calc);

azimuth_current := AzimuthElevationControl.act_position;
elevation_current := ElevationControl.act_position;

hor2eq(alt := elevation_current, 
		az := azimuth_current,
		jd := jd,
		lat := latitude,
		lon := longitude,
		altitude := altitude,
		ra => rightascension_calc,
		dec => declination_calc);		

sunpos(JD := jd);
sunhor2(alpha := sunpos.ra,
		delta := sunpos.Dec,
		lon := longitude,
		lat := latitude,
		JD := jd + time_offset);
solz := 90.0 - sunhor2.alt;
		
// TODO check sign; offset is applied later
derotation_calc := F_DerotatorPosition2(azimuth_calc, elevation_calc, declination_calc, latitude);
IF Tracking THEN
	DerotatorVelocity := F_Derotatorvelocity(elevation_calc, azimuth_calc, latitude);
ELSE
	DerotatorVelocity := 10.0;
END_IF
		
poweronwarning(IN := power OR (NOT ElevationControl.enable AND HydraulicsControl.brake_open), PT := T#250MS);
powerontrigger(CLK := power);
powerofftrigger(CLK := power);
poweron_reset(IN := power AND NOT PendantControl.manual, PT := T#50MS);
// park the telescope after 12 hours
power_timeout(IN := power, PT := T#12H);
IF power_timeout.Q THEN
	power := FALSE;
END_IF
// reset fan
FanControl.reset := poweron_reset.Q OR reset;
CoverControl.reset := poweron_reset.Q OR reset;

IF Nasmyth_port = 1 THEN
	NasmythControl.right := FALSE;
	IF NasmythControl.Nasmyth_left THEN
		NasmythControl.left := FALSE;
		NasmythControl.enable := FALSE;
	ELSE
		NasmythControl.left := TRUE;
		NasmythControl.enable := TRUE;
	END_IF
ELSIF Nasmyth_port = 2 THEN
	NasmythControl.left := FALSE;
    IF NasMythControl.Nasmyth_right THEN
		NasmythControl.right := FALSE;
		NasmythControl.enable := FALSE;
	ELSE
		NasmythControl.right := TRUE;
		NasmythControl.enable := TRUE;
	END_IF
ELSE
	NasmythControl.right := FALSE;
	NasmythControl.left := FALSE;
	NasmythControl.enable := FALSE;	
END_IF
	
IF power THEN
	poweron();
//ELSE
	//poweroff();
END_IF
(*
IF NOT power AND NOT PendantControl.manual THEN
	// if the power is deactivatied and we are on automatic, ...
	IF CoverControl.isclosed THEN
		// if the covers are closed, disable them
		CoverControl.close := FALSE;
		CoverControl.enable := FALSE;
(*	ELSIF Environment.WeatherBad THEN
		// if the covers are not closed and the weather is bad, close them
		CoverControl.enable := TRUE;
		CoverControl.close := TRUE; *)
	END_IF
END_IF
*)		
// set TCS_command according to state variables ordered by precedence
IF track THEN
	TCS_command := E_TCSCommand.track;
	goto := FALSE;
	slew := FALSE;
ELSIF goto THEN
	TCS_command := E_TCSCommand.goto;
	track := FALSE;
	slew := FALSE;
ELSIF gohome THEN
	TCS_command := E_TCSCommand.gohome;
	goto := FALSE;
	track := FALSE;
	slew := FALSE;
ELSIF slew THEN
	TCS_command := E_TCSCommand.slew;
	goto := FALSE;
	track := FALSE;
ELSIF park THEN
	TCS_command := E_TCSCommand.park;
	goto := FALSE;
	track := FALSE;
	slew := FALSE;
ELSIF pumping THEN
	TCS_command := E_TCSCommand.pumping;
ELSIF stop THEN
	TCS_command := E_TCSCommand.stop;
	goto := FALSE;
	track := FALSE;
	slew := FALSE;
	gohome := FALSE;
	park := FALSE;
ELSE
	TCS_command := E_TCSCommand.no_command;
	ElevationControl.MoveAxis := FALSE;
	AzimuthElevationControl.MoveAxis := FALSE;
END_IF

IF NOT track THEN
	ElevationControl.Tracking := FALSE;
	AzimuthElevationControl.Tracking := FALSE;
	DerotatorControl.Tracking := FALSE;
END_IF

IF TCS_command = E_TCSCommand.park THEN
	IF parktelescope() THEN
		power := FALSE;
	END_IF
ELSIF TCS_command = E_TCSCommand.gohome THEN
	IF hometelescope() THEN
		gohome := FALSE;
	END_IF
ELSIF TCS_command = E_TCSCommand.track THEN
	ElevationControl.position := elevation_calc + elevation_offset;
	AzimuthElevationControl.position := azimuth_calc + azimuth_offset;
	DerotatorControl.position := derotation_calc + derotator_offset;
	DerotatorControl.Velocity := DerotatorVelocity;
	ElevationControl.Tracking := TRUE;
	AzimuthElevationControl.Tracking := TRUE;
	DerotatorControl.Tracking := TRUE;
	
ELSIF TCS_command = E_TCSCommand.goto THEN
	gototelescope();
ELSIF TCS_command = E_TCSCommand.slew THEN
	slewtelescope();
ELSIF TCS_command = E_TCSCommand.pumping THEN
	gotopumping();
END_IF
 
sliding := ElevationControl.MoveAxis OR 
			AzimuthElevationControl.MoveAxis OR
			DerotatorControl.MoveAxis;
			
tracking := ElevationControl.Tracking AND 
			AzimuthElevationControl.Tracking AND
			DerotatorControl.Tracking;
			
stopped :=  ElevationControl.ElevationAxis.StandStill AND 
			AzimuthElevationControl.AzimuthAxis.StandStill AND
			DerotatorControl.DerotatorAxis.StandStill;
			
homed := ElevationControl.Calibrated AND
			AzimuthElevationControl.calibrated AND
			FilterWheelControl.Calibrated AND
			FocusControl.Calibrated AND
			DerotatorControl.Calibrated;
			
ready := homed AND CoverControl.isopen AND HydraulicsControl.brake_open AND NOT error;

IF NOT error THEN
	reset := FALSE;
END_IF

GVL_Telescope.horn := poweronwarning.Q OR Pendantcontrol.horn;

MQTTTimer(IN:=TRUE);
IF MQTTTimer.Q THEN // publish new payload every second
	MQTTTimer(IN:=FALSE);

	MAIN.MQTTClient.Publish('telescope', 'dome', 'Azimuth', LREAL_TO_FMTSTR(azimuth_current, 5, TRUE));
	MAIN.MQTTClient.Publish('telescope', 'dome', 'Elevation', LREAL_TO_FMTSTR(elevation_current, 5, TRUE));
	MAIN.MQTTClient.Publish('telescope', 'dome', 'HourAngle', LREAL_TO_FMTSTR(hourangle_calc, 5, TRUE));
	MAIN.MQTTClient.Publish('telescope', 'dome', 'RightAscension', LREAL_TO_FMTSTR(rightascension_calc, 5, TRUE));
	MAIN.MQTTClient.Publish('telescope', 'dome', 'Declination', LREAL_TO_FMTSTR(declination_calc, 5, TRUE));
	MAIN.MQTTClient.Publish('telescope', 'dome', 'Derotator', LREAL_TO_FMTSTR(derotation_calc, 5, TRUE));
	MAIN.MQTTClient.Publish('telescope', 'dome', 'errorid',		UDINT_TO_STRING(errorid));
	MAIN.MQTTClient.Publish('telescope', 'dome', 'error',		BOOL_TO_STRING(error));
	MAIN.MQTTClient.Publish('telescope', 'dome', 'ready',		BOOL_TO_STRING(ready));
	MAIN.MQTTClient.Publish('telescope', 'dome', 'sliding',		BOOL_TO_STRING(sliding));
	MAIN.MQTTClient.Publish('telescope', 'dome', 'tracking', 	BOOL_TO_STRING(tracking));
	MAIN.MQTTClient.Publish('telescope', 'dome', 'stopped',		BOOL_TO_STRING(stopped));
	MAIN.MQTTClient.Publish('telescope', 'dome', 'homed',		BOOL_TO_STRING(homed));
END_IF

StatusWord.0 := error;
StatusWord.1 := ready;
StatusWord.2 := sliding;
StatusWord.3 := tracking;
StatusWord.4 := stopped;
StatusWord.5 := homed;

IF StatusWord<>LastStatus THEN // publish new payload every second
	LastStatus := StatusWord;
	MAIN.MQTTClient.Publish('telescope', 'dome', 'error',		BOOL_TO_STRING(error));
	MAIN.MQTTClient.Publish('telescope', 'dome', 'ready',		BOOL_TO_STRING(ready));
	MAIN.MQTTClient.Publish('telescope', 'dome', 'sliding',		BOOL_TO_STRING(sliding));
	MAIN.MQTTClient.Publish('telescope', 'dome', 'tracking', 	BOOL_TO_STRING(tracking));
	MAIN.MQTTClient.Publish('telescope', 'dome', 'stopped',		BOOL_TO_STRING(stopped));
	MAIN.MQTTClient.Publish('telescope', 'dome', 'homed',		BOOL_TO_STRING(homed));
END_IF


(* Event function blocks start here. *)
TCSpowerEvent(	Trigger := powerfailure, 
				Level := ADSLOG_MSGTYPE_ERROR,
				FormatString := 'power %s',
				OnMessage := 'Failure',
				OffMessage := 'OK');

TCSgohomeEvent(	Trigger := gohome, 
				Level := ADSLOG_MSGTYPE_HINT,
				FormatString := 'GOHOME %s',
				OnMessage := 'commencing',
				OffMEssage := 'completed');
TCSparkEvent(	Trigger := park, 
				Level := ADSLOG_MSGTYPE_HINT,
				FormatString := 'PARK %s',
				OnMessage := 'commencing',
				OffMEssage := 'completed');
TCSgotoEvent(	Trigger := goto, 
				Level := ADSLOG_MSGTYPE_HINT,
				FormatString := 'GOTO %s',
				OnMessage := 'commencing',
				OffMEssage := 'completed');
TCStrackEvent(	Trigger := track, 
				Level := ADSLOG_MSGTYPE_HINT,
				FormatString := 'TRACK %s',
				OnMessage := 'commencing',
				OffMEssage := 'completed');
TCSstopEvent(	Trigger := stop, 
				Level := ADSLOG_MSGTYPE_WARN,
				FormatString := 'STOP %s',
				OnMessage := 'commencing',
				OffMEssage := 'completed',
				OffLevel := ADSLOG_MSGTYPE_HINT);
AltitudeEvent(	Trigger := power AND elevation_calc<0.0, 
				Level := ADSLOG_MSGTYPE_WARN,
				FormatString := '%s',
				OnMessage := 'Target below horizon',
				OffMEssage := '');
TCSreadyEvent(	Trigger := power AND ready, 
				Level := ADSLOG_MSGTYPE_HINT,
				FormatString := '%s',
				OnMessage := 'RoboTel startup finished');

METHOD gotopumping : BOOL
VAR_INPUT
END_VAR
ElevationControl.position := elevation;
ElevationControl.MoveAxis := TRUE;
AzimuthElevationControl.position := azimuth;
AzimuthElevationControl.MoveAxis := TRUE;
DerotatorControl.position := 90.0;
DerotatorControl.MoveAxis := TRUE;

IF ElevationControl.ElevationAxis.StopDone AND 
	AzimuthElevationControl.AzimuthAxis.StopDone AND 
	DerotatorControl.DerotatorAxis.StopDone THEN
	ElevationControl.MoveAxis := FALSE;
	AzimuthElevationControl.MoveAxis := FALSE;
	DerotatorControl.MoveAxis := FALSE;
	pumping := FALSE;
	gotopumping := TRUE;
ELSE
	gotopumping := FALSE;
END_IF
END_METHOD

METHOD gototelescope : BOOL
VAR_INPUT
END_VAR
ElevationControl.position := elevation_calc + elevation_offset;
ElevationControl.MoveAxis := TRUE;
AzimuthElevationControl.position := azimuth_calc + azimuth_offset;
AzimuthElevationControl.MoveAxis := TRUE;
DerotatorControl.position := derotation_calc + derotator_offset;
DerotatorControl.MoveAxis := TRUE;
IF ElevationControl.ElevationAxis.MoveDone AND 
	AzimuthElevationControl.AzimuthAxis.MoveDone AND
	DerotatorControl.DerotatorAxis.MoveDone THEN
	ElevationControl.MoveAxis := FALSE;
	AzimuthElevationControl.MoveAxis := FALSE;
	DerotatorControl.MoveAxis := FALSE;
	goto := FALSE;
	gototelescope := TRUE;
ELSE
	gototelescope := FALSE;
END_IF
END_METHOD

METHOD hometelescope : BOOL
VAR_INPUT
END_VAR

VAR
	HomeEvent: FB_Eventlog;
END_VAR
ElevationControl.position := elevation_home;
ElevationControl.MoveAxis := TRUE;
AzimuthElevationControl.position := azimuth_home;
AzimuthElevationControl.MoveAxis := TRUE;
IF ElevationControl.ElevationAxis.MoveDone AND 
	AzimuthElevationControl.AzimuthAxis.MoveDone THEN
	gohome := FALSE;
	hometelescope := TRUE;
ELSE
	hometelescope := FALSE;
END_IF

HomeEvent(Trigger := hometelescope, 
			Level := ADSLOG_MSGTYPE_HINT,
			FormatString := '%s',
			OnMessage := 'Telescope is homed.');
END_METHOD

METHOD parktelescope : BOOL
VAR_INPUT
END_VAR


VAR
	ParkEvent: FB_Eventlog;
END_VAR
gohome := 	FALSE;
track := 	FALSE;
goto := 	FALSE;
slew := 	FALSE;
pumping :=	FALSE;

ElevationControl.position := elevation_park;
AzimuthElevationControl.position := azimuth_park;
ElevationControl.MoveAxis := TRUE;
AzimuthElevationControl.MoveAxis := TRUE;
CoverControl.close := TRUE;
IF ElevationControl.ElevationAxis.MoveDone AND 
	AzimuthElevationControl.AzimuthAxis.MoveDone AND 
	CoverControl.isclosed THEN
	park := FALSE;
	parktelescope := TRUE;
ELSE
	parktelescope := FALSE;
END_IF

ParkEvent(Trigger := parktelescope, 
			Level := ADSLOG_MSGTYPE_HINT,
			FormatString := '%s',
			OnMessage := 'Telescope is parked.');
END_METHOD

METHOD poweroff : BOOL
VAR_INPUT
END_VAR
VAR
	power_is_off: 	BOOL;
	offtrigger:		R_TRIG;
	PowerOffEvent: 	FB_Eventlog;
END_VAR
gohome := 	FALSE;
park  := 	FALSE;
track := 	FALSE;
goto := 	FALSE;
slew := 	FALSE;
pumping :=	FALSE;
// disable azimuth
// disbale elevation (closes brake)
IF stopped THEN
	AzimuthElevationControl.enable := FALSE;
	ElevationControl.enable := FALSE;
END_IF
// disable Focus
(*
IF FocusControl.FocusAxis.StandStill THEN
	Focuscontrol.enable := FALSE;
END_IF
*)
// disable filterwheel
FilterWheelControl.Enable := FALSE;
// disable derotator
DerotatorControl.enable := FALSE;

IF NOT ElevationControl.enable THEN
	// disable hydraulics
	HydraulicsControl.close_brake := TRUE;
	HydraulicsControl.stop := TRUE;
END_IF

IF HydraulicsControl.brake_closed THEN
	// close cover
	CoverControl.close := TRUE;	
END_IF

power_is_off := NOT power 
	AND NOT AzimuthElevationControl.enable 
	AND NOT ElevationControl.enable 
//	AND NOT FocusControl.enable
	AND NOT FilterWheelControl.Enable
	AND NOT DerotatorControl.enable
	AND HydraulicsControl.brake_closed
	AND CoverControl.isclosed;

poweroff := power_is_off;

offtrigger(CLK := power_is_off);
	
PowerOffEvent(Trigger := FALSE, 
				Level := ADSLOG_MSGTYPE_HINT,
				FormatString := '%s',
				OnMessage := 'RoboTel shutdown finished');
END_METHOD

METHOD poweron : BOOL
VAR_INPUT
END_VAR
VAR
END_VAR
IF NOT Main.brake_clearing THEN
	powerfailure := TRUE;
	TCSpowerEvent.OnMessage := 'failure: brake clearing not set';
	power := FALSE;
ELSIF NOT Transformer.power_OK THEN
	powerfailure := TRUE;
	TCSpowerEvent.OnMessage := 'failure: main power failure';
	power := FALSE;
ELSIF NOT Main.phase_available THEN
	powerfailure := TRUE;
	TCSpowerEvent.OnMessage := 'failure: hydraulics power failure';
	power := FALSE;
ELSE
	powerfailure := FALSE;		
END_IF
// enable hydraulics
HydraulicsControl.start := TRUE;
// open cover
// COVER MUST BE OPENED FOR A SUCCESSFUL WAKE & SHAKE COMMAND!
CoverControl.enable := TRUE;
//CoverControl.reset := poweron_reset.Q;
Covercontrol.open := TRUE;
IF Covercontrol.isopen THEN
	Covercontrol.open := FALSE;
END_IF
// enable elevation enable azimuth

IF MAIN.ready AND CoverControl.isopen THEN
	HydraulicsControl.open_brake := TRUE;
	ElevationControl.enable := TRUE;
	AzimuthElevationControl.enable := TRUE;
END_IF

IF ElevationControl.Ready AND NOT ElevationControl.Calibrated THEN
	ElevationControl.HomeAxis := TRUE;
END_IF

IF AzimuthElevationControl.ready AND NOT AzimuthElevationControl.calibrated THEN
	AzimuthElevationControl.HomeAxis := TRUE;
END_IF

// if the dome is not calibrated while the power is on, start calibration
IF NOT DomeControl.Calibrated THEN
	DomeControl.HomeAxis := TRUE;
ELSE
	DomeControl.HomeAxis := FALSE;
END_IF

// enable derotator
IF ElevationControl.Ready THEN
	DerotatorControl.enable := TRUE;
	DerotatorControl.HomeAxis := DerotatorControl.Ready AND NOT DerotatorControl.Calibrated;
END_IF

// enable filterwheel after Derotator Axis to avoid additional torque
IF DerotatorControl.Calibrated THEN
	FilterWheelControl.Enable := TRUE;
	FilterWheelControl.HomeAxis := NOT FilterWheelControl.Calibrated;
END_IF

// enable focus
FocusControl.enable := TRUE;
IF FocusControl.ready AND NOT FocusControl.Calibrated THEN
	FocusControl.HomeAxis := TRUE;
END_IF
FocusDelay(IN := FocusControl.Calibrated AND FocusControl.Ready);
IF FocusDelay.Q THEN
	FocusControl.position := focus_position;
	FocusControl.MoveAxis := ABS(FocusControl.actual_position - focus_position) > 0.005;
END_IF
END_METHOD

METHOD slewtelescope : BOOL
VAR_INPUT
END_VAR
ElevationControl.position := elevation;
ElevationControl.MoveAxis := TRUE;
AzimuthElevationControl.position := azimuth;
AzimuthElevationControl.MoveAxis := TRUE;
DerotatorControl.position := elevation + derotator_offset;
DerotatorControl.MoveAxis := TRUE;
IF ElevationControl.ElevationAxis.MoveDone 
	AND AzimuthElevationControl.AzimuthAxis.MoveDone 
	AND DerotatorControl.DerotatorAxis.MoveDone THEN
	ElevationControl.MoveAxis := FALSE;
	AzimuthElevationControl.MoveAxis := FALSE;
	DerotatorControl.MoveAxis := FALSE;
	slew := FALSE;
	slewtelescope := TRUE;
ELSE
	slewtelescope := FALSE;
END_IF
END_METHOD

END_PROGRAM

// ---- POUs/FunctionBlocks/FB_AstroClock.TcPOU
FUNCTION_BLOCK FB_AstroClock
VAR_INPUT
END_VAR
VAR_OUTPUT
        time_RTCEX      : DT;
        time_RTCEX2     : TIMESTRUCT;
        nMilliseconds   : DWORD;
        nMicroseconds   : DWORD;
END_VAR
VAR
	        fbGetLocalTime  : NT_GetTime;
        bBusy           : BOOL;
        bError          : BOOL;
        nErrID          : UDINT;
        presetTime      : TIMESTRUCT;

        syncTimer       : TON;
        syncTrigger     : F_TRIG;
        bSynchronize    : BOOL;

        fbRTC           : RTC;
        bValid_RTC      : BOOL;
        time_RTC        : DT;

        fbRTC_EX        : RTC_EX;
        bValid_RTCEX    : BOOL;

        fbRTC_EX2       : RTC_EX2;
        bValid_RTCEX2   : BOOL;
END_VAR

(*
TYPE TIMESTRUCT
STRUCT
   wYear            : WORD;
   wMonth           : WORD;
   wDayOfWeek       : WORD;
   wDay             : WORD;
   wHour            : WORD;
   wMinute          : WORD;
   wSecond          : WORD;
   wMilliseconds    : WORD;
END_STRUCT
END_TYPE
*)

syncTimer(IN := NOT SyncTimer.Q, PT := T#5S);
fbGetLocalTime(START := syncTimer.Q,
	TMOUT := DEFAULT_ADS_TIMEOUT,
	Busy => bBusy,
	ERR => bError,
	ERRID => nErrID,
	TIMESTR => presetTime);

syncTrigger(CLK := bBusy AND NOT bError, Q => bSynchronize);

fbRTC(EN := bSynchronize,
	PDT := SYSTEMTIME_TO_DT(presetTime),
	Q => bValid_RTC,
	CDT => time_RTC);
	
fbRTC_EX(EN := bSynchronize,
	PDT := SYSTEMTIME_TO_DT(presetTime),
	PMSEK := presetTime.wMilliseconds,
	Q => bValid_RTCEX,
	CDT => time_RTCEX,
	CMSEK => nMilliseconds);

fbRTC_EX2(EN := bSynchronize,
	PDT := presetTime,
	PMICRO := 0,
	Q => bValid_RTCEX2,
	CDT => time_RTCEX2,
	CMICRO => nMicroseconds);

END_FUNCTION_BLOCK

// ---- POUs/FunctionBlocks/FB_EQ2HOR2.TcPOU
FUNCTION_BLOCK FB_EQ2HOR2
VAR_INPUT
	// right ascension in degrees
	alpha: LREAL;
	// declination in degrees
	delta: LREAL;
	// longitude in degrees
	lon: LREAL;
	// latitude in degrees
	lat: LREAL;
	// Julian Days
	JD: LREAL;
END_VAR
VAR_OUTPUT
	// altitude in degrees
	alt: LREAL;
	// azimuth in degrees
	az: LREAL;
	// hour angle in degreesss
	ha: LREAL;
END_VAR
VAR
	lst, 
	T , theta0, gmst: LREAL;
	// helper variables
	sinalt, sinaz, cosaz, cosalt, az1, az2, az3, length,
	// in radians
	phi_r, tau_r, alpha_r, delta_r: LREAL;
	//quadrant: UINT;
END_VAR
VAR CONSTANT
	d2r:	LREAL := PI/180.0;
	r2d:	LREAL := 180.0/PI;
	//h2r:	LREAL := PI/12.0;
	//h2d:	LREAL := 15.0;
END_VAR

(* 
source: http://star-www.st-and.ac.uk/~fv/webnotes/chapter7.htm
https://squarewidget.com/astronomical-calculations-sidereal-time/

*)
//lst := ct2lst(lon, jd);
T := ((JD - 2451545.0) / 36525.0);
theta0 := 280.46061837 + 360.98564736629 * (JD - 2451545.0) + (0.000387933 * T * T) - (T * T * T / 38710000.0); // (12.4)
gmst := MODABS(theta0, 360.0);
lst := gmst + lon; // LST in degrees
// ha := MODABS(lst*15.0 - alpha, 360.0);
ha := MODABS(lst - alpha, 360.0);

alpha_r := alpha * d2r;
delta_r := delta * d2r;
tau_r := lst*d2r - alpha_r;
//tau_r := MODABS(lst*d2r - alpha_r, 2.0*PI);
phi_r := lat*d2r;

//sinalt := (SIN(delta*d2r)*SIN(lat*d2r)) + (COS(delta*d2r)*COS(lat*d2r)*COS(ha*d2r));
sinalt := SIN(phi_r)*SIN(delta_r) + COS(phi_r)*COS(delta_r)*COS(tau_r);
alt := ASIN(sinalt) * r2d;
cosalt := COS(alt*d2r);

IF ABS(cosalt) > 0.0 THEN
	sinaz := -SIN(tau_r)*COS(delta_r)/cosalt;
ELSE
	sinaz := 0.0;
END_IF

IF ABS(cosalt*COS(phi_r)) > 0.0 THEN
	cosaz := (SIN(delta_r) - SIN(phi_r)*sinalt)
			/(cosalt*COS(phi_r));
ELSE
	cosaz := 0.0;
END_IF

length := sinaz*sinaz + cosaz*cosaz;

az1 := ASIN(LIMIT(-1.0, sinaz, 1.0)) * r2d;

az2 := ACOS(LIMIT(-1.0, cosaz, 1.0)) * r2d;

az3 := ATAN2(SIN(phi_r)*COS(tau_r) - COS(phi_r)*TAN(delta_r), SIN(tau_r)) * r2d;

IF sinaz >= 0.0 AND cosaz >=0.0 THEN // Q I
	az := az1;
ELSIF sinaz < 0.0 AND cosaz >= 0.0 THEN // Q II
	az := MODABS(-az2, 360.0);
ELSIF sinaz < 0.0 AND cosaz < 0.0 THEN // Q III
	az := 180 - az1;
ELSIF sinaz >= 0.0 AND cosaz < 0.0 THEN // Q IV
	az := az2;
END_IF

END_FUNCTION_BLOCK

// ---- POUs/Functions/ATAN2.TcPOU
FUNCTION ATAN2 : LREAL // result in radians
VAR_INPUT
	y, x: LREAL;
END_VAR
VAR
END_VAR

(* source: https://de.wikipedia.org/wiki/Arctan2 *)
ATAN2 := 0.0;

IF x > 0 THEN
	ATAN2 := ATAN(y/x);
ELSIF x < 0 AND y > 0 THEN
	ATAN2 := ATAN(y/x) + PI;
ELSIF x < 0 AND y = 0 THEN
	ATAN2 := PI;
ELSIF x < 0 AND y < 0 THEN
	ATAN2 := ATAN(y/x) - PI;
ELSIF x = 0 AND y > 0 THEN
	ATAN2 := PI/2.0;
ELSIF x = 0 AND y < 0 THEN
	ATAN2 := -PI/2.0;
END_IF

END_FUNCTION

// ---- POUs/FunctionBlocks/FB_HOR2EQ.TcPOU
FUNCTION_BLOCK FB_HOR2EQ
VAR_INPUT
	//altitude (in degrees) [scalar OR vector]
	alt: LREAL;  
	//azimuth angle (in degrees, measured EAST from NORTH, but see keyword WS below.) [scalar or vector]
	az: LREAL;
	// Julian Date [scalar or vector], double precision
	JD: LREAL;
	lat:	LREAL;
	lon:	LREAL;
	WS:	BOOL;
	precess:	BOOL := TRUE;
	NUTATE:		BOOL := TRUE;
	aberration:	BOOL := TRUE;
	refract:	BOOL := TRUE;
	altitude:	LREAL := 0.0;
END_VAR
VAR_OUTPUT
	// Right Ascension of object  (J2000) in degrees (FK5)
	ra: 	LREAL;
	// Declination of object (J2000) in degrees (FK5)
	dec:	LREAL;
	// hour angle (in degrees) (optional)
	ha:		LREAL;
END_VAR
VAR
	
	alt_,
	az_,
	lmst,
	J_now: LREAL;
	co_nutate: 		FB_CO_NUTATE;
	co_aberration: 	CO_ABERRATION;
	co_refract:		CO_REFRACT;
	fbprecess:		FB_PRECESS;
	altaz2hadec:	FB_ALTAZ2HADEC;
	last: LREAL;
	dra1: LREAL;
	ddec1: LREAL;
	eps: LREAL;
	d_psi: LREAL;
	dra2: LREAL;
	ddec2: LREAL;
END_VAR
VAR CONSTANT
	//d2r:	LREAL := PI/180.0;
	//r2d:	LREAL := 180.0/PI;
	//h2r:	LREAL := PI/12.0;
	h2d:	LREAL := 15.0;
END_VAR



alt_ := alt;   //do this so we don't change ra, dec arrays.
az_ := az;


//*******************************************************************************************
// Make Correction for ATMOSPHERIC REFRACTION
// (use this for visible and radio wavelengths; author is unsure about other wavelengths)
IF refract THEN 
	co_refract(	old_alt := alt, 
				altitude := altitude, 
				to_observed := TRUE, 
				new_alt => alt);
END_IF

IF WS THEN 
	az_ := az_ - 180.0;
END_IF

co_nutate(	jd := jd, 
			ra := 45.0, 
			dec := 45.0, 
			d_ra => dra1, 
			d_dec => ddec1, 
			eps => eps, 
			d_psi => d_psi);
//******************************************************************************
//Calculate LOCAL APPARENT SIDEREAL TIME
// first get local mean sidereal time (lmst)
// get LST (in hours) - note:this is indep of tzone since giving jd
lmst := ct2lst( lon, jd);
// convert LMST TO degrees (btw, THIS is the RA OF the zenith)
lmst := lmst*h2d;
// calculate local APPARENT sidereal time (last)
// ADD correction in degrees
last := lmst + d_psi *COS(eps)/3600.0 ; 

//****************************************************************************
// Now do the spherical trig to get APPARENT Hour Angle [degrees], and
// declination [degrees].
altaz2hadec( alt := alt_, az := az_, lat := lat, ha => ha, dec => dec);

// Find Right Ascension (in degrees, from 0 to 360.)
 ra := MODABS(last - ha + 360.0, 360.0);



//*****************************************************************************
// calculate NUTATION and ABERRATION Corrections to Ra-Dec
IF NUTATE THEN
	co_nutate(	jd := jd, 
			ra := ra, 
			dec := dec, 
			d_ra => dra1, 
			d_dec => ddec1, 
			eps => eps, 
			d_psi => d_psi);
ELSE
	dra1 := 0.0;
	ddec1 := 0.0;	
END_IF
IF aberration THEN
	co_aberration(	jd := jd, 
				ra := ra, 
				dec := dec, 
				d_ra => dra2, 
				d_dec => ddec2, 
				eps := eps);
ELSE
	dra2 := 0.0;
	ddec2 := 0.0;	
END_IF
//******************************************************************************
// Make Nutation and Aberration Corrections (if wanted)

ra := ra - (dra1 + dra2)/3600.0;
dec := dec - (ddec1 + ddec2)/3600.0;
 //compute current equinox
J_now := (JD - 2451545.0)/365.25 + 2000.0 ;

//*****************************************************************************
// PRECESS coordinates to current date
// (uses astro lib procedure PRECESS.pro)

IF precess THEN 
	fbprecess( ra := ra, dec := dec, 
	EQUINOX1 := 2000.0, EQUINOX2 := J_now, 
	ra_precessed =>ra, dec_precessed => dec);                   
END_IF

END_FUNCTION_BLOCK

// ---- POUs/FunctionBlocks/FB_CO_NUTATE.TcPOU
FUNCTION_BLOCK FB_CO_NUTATE
VAR_INPUT
	jd,
	ra,
	dec:	LREAL;
END_VAR
VAR_OUTPUT
	d_ra,
	d_dec,
	eps,
	d_psi,
	d_eps:	LREAL;
END_VAR
VAR
	T, 
	eps0,
ce, se,x,y,z,x2,y2,z2,rad,xyproj,ra2,dec2: LREAL;
	nutate:	FB_NUTATE;
END_VAR
VAR CONSTANT
	d2r:	LREAL := PI/180.0;
	d2as:	LREAL := PI/(180.0*3600.0);
END_VAR

// Julian centuries FROM J2000 OF jd.
T := (jd -2451545.0)/36525.0; 

// must calculate obliquity OF ecliptic
nutate(jd := jd,
		nut_long => d_psi, 
		nut_obliq => d_eps); 

eps0 := 23.4392911*3600.0 - 46.8150*T - 0.00059*EXPT(T, 2) + 0.001813*EXPT(T, 3);
eps := (eps0 + d_eps)/3600.0*d2r; // TRUE obliquity OF the ecliptic in radians
 
//useful numbers
ce := COS(eps);
se := SIN(eps);

// convert ra-dec to equatorial rectangular coordinates
x := COS(ra*d2r) * COS(dec*d2r);
y := SIN(ra*d2r) * COS(dec*d2r);
z := SIN(dec*d2r);

// apply corrections to each rectangular coordinate
x2 := x - (y*ce + z*se)*d_psi * d2as;
y2 := y + (x*ce*d_psi - z*d_eps) * d2as;
z2 := z + (x*se*d_psi + y*d_eps) * d2as;

// convert back to equatorial spherical coordinates
rad := SQRT(x2*x2 + y2*y2 + z2*z2);
xyproj := SQRT(x2*x2 + y2*y2);

ra2  := x2 * 0.0;
dec2 := x2 * 0.0;

// Calculate Ra and Dec in RADIANS (later convert to DEGREES)
IF (xyproj = 0) AND (z <> 0) THEN
	// places where xyproj=0 (point at NCP or SCP)
	dec2 := ASIN(z2/rad);
	ra2 := 0.0;
END_IF
 
IF (xyproj <> 0) THEN
	// places other than NCP or SCP
	ra2 := ATAN2(y2, x2);
	dec2 := ASIN(z2/rad);
END_IF

// convert to DEGREES

ra2 := ra2 /d2r;
dec2 := dec2 /d2r;

ra2 := MODABS(ra2, 360.0);


// Return changes in ra and dec in arcseconds
d_ra := (ra2 - ra) * 3600.0;
d_dec := (dec2 - dec) * 3600.0;

END_FUNCTION_BLOCK

// ---- POUs/FunctionBlocks/FB_NUTATE.TcPOU
FUNCTION_BLOCK FB_NUTATE
VAR_INPUT
	jd:	LREAL;
END_VAR
VAR_OUTPUT
	nut_long, nut_obliq: LREAL := 0.0;
END_VAR
VAR
	t: LREAL;
	d, M, Mprime, F, omega: LREAL;
	arg, sarg, carg:  ARRAY[0..62] OF LREAL;
	I: INT;
END_VAR
VAR CONSTANT
	dtor:	LREAL := PI/180.0;
	coeff1:	ARRAY[0..3] OF LREAL := [297.85036, 445267.111480, -0.0019142,  1.0/189474];
	coeff2:	ARRAY[0..3] OF LREAL := [357.52772,  35999.050340, -0.0001603, -1.0/3E5]; 
	coeff3:	ARRAY[0..3] OF LREAL := [134.96298, 477198.867398,  0.0086972,  1.0/5.625E4]; 
	coeff4:	ARRAY[0..3] OF LREAL :=  [93.27191, 483202.017538, -0.0036825, -1.0/3.27270E5]; 
  	coeff5: ARRAY[0..3] OF LREAL := [125.04452,  -1934.136261,  0.0020708,  1.0/4.5E5];
	d_lng: ARRAY[0..62] OF LREAL := [0,-2,0,0,0,0,-2,0,0,-2,-2,-2,0,2,0,2,0,0,-2,0,2,0,0,-2,0,-2,0,0,2,-2,0,-2,0,0,2,2,0,-2,0,2,2,-2,-2,2,2,0,-2,-2,0,-2,-2,0,-1,-2,1,0,0,-1,0,0,2,0,2]; 
	m_lng: ARRAY[0..62] OF LREAL := [0,0,0,0,1,0,1,0,0,-1,17(0),2,0,2,1,0,-1,0,0,0,1,1,-1,0,0,0,0,0,0,-1,-1,0,0,0,1,0,0,1,0,0,0,-1,1,-1,-1,0,-1];
	mp_lng: ARRAY[0..62] OF LREAL := [0,0,0,0,0,1,0,0,1,0,1,0,-1,0,1,-1,-1,1,2,-2,0,2,2,1,0,0,-1,0,-1,0,0,1,0,2,-1,1,0,1,0,0,1,2,1,-2,0,1,0,0,2,2,0,1,1,0,0,1,-2,1,1,1,-1,3,0];
	f_lng: ARRAY[0..62] OF LREAL := [0,2,2,0,0,0,2,2,2,2,0,2,2,0,0,2,0,2,0,2,2,2,0,2,2,2,2,0,0,2,0,0,0,-2,2,2,2,0,2,2,0,2,2,0,0,0,2,0,2,0,2,-2,0,0,0,2,2,0,0,2,2,2,2];
	om_lng: ARRAY[0..62] OF LREAL := [1,2,2,2,0,0,2,1,2,2,0,1,2,0,1,2,1,1,0,1,2,2,0,2,0,0,1,0,1,2,1,1,1,0,1,2,2,0,2,1,0,2,1,1,1,0,1,1,1,1,1,0,0,0,0,0,2,0,0,2,2,2,2];
	sin_lng: ARRAY[0..62] OF LREAL := [-171996, -13187, -2274, 2062, 1426, 712, -517, -386, -301, 217, -158, 129, 123, 63, 63, -59, -58, -51, 48, 46, -38, -31, 29, 29, 26, -22, 21, 17, 16, -16, -15, -13, -12, 11, -10, -8, 7, -7, -7, -7, 6,6,6,-6,-6,5,-5,-5,-5,4,4,4,-4,-4,-4,3,-3,-3,-3,-3,-3,-3,-3 ];
	sdelt: ARRAY[0..62] OF LREAL := [-174.2, -1.6, -0.2, 0.2, -3.4, 0.1, 1.2, -0.4, 0, -0.5, 0, 0.1, 0,0,0.1, 0,-0.1,10(0), -0.1, 0, 0.1, 33(0)];
	cos_lng: ARRAY[0..62] OF LREAL := [ 92025, 5736, 977, -895, 54, -7, 224, 200, 129, -95,0,-70,-53,0, -33, 26, 32, 27, 0, -24, 16,13,0,-12,0,0,-10,0,-8,7,9,7,6,0,5,3,-3,0,3,3, 0,-3,-3,3,3,0,3,3,3, 14(0)] ;
	cdelt: ARRAY[0..62] OF LREAL := [8.9, -3.1, -0.5, 0.5, -0.1, 0.0, -0.6, 0.0, -0.1, 0.3, 53(0)];
END_VAR

//  form time in Julian centuries from 1900.0

t := (jd - 2451545.0)/36525.0;

// Mean elongation of the Moon

d := poly(T, coeff1)*dtor;
d := MODABS(d, 2.0*PI);

// Sun's mean anomaly

M := poly(T,coeff2)*dtor;
M := MODABS(M, 2.0*PI);

// Moon's mean anomaly

Mprime := poly(T,coeff3)*dtor;
Mprime := MODABS(Mprime, 2.0*PI);

// Moon's argument of latitude

F := poly(T, coeff4 )*dtor;
F := MODABS(F, 2.0*PI);

// Longitude OF the ascending node OF the Moon's mean orbit on the ecliptic,
//  measured from the mean equinox of the date

omega := poly(T, coeff5)*dtor;
omega := MODABS(omega, 2.0*PI);


// Sum the periodic terms 
FOR i:=0 TO 62 DO
	arg[i] := d_lng[i]*d + m_lng[i]*m +mp_lng[i]*mprime + f_lng[i]*f +om_lng[i]*omega;
	sarg[i] := SIN(arg[i]);
	carg[i] := COS(arg[i]);
END_FOR

